LIN {X 0,Y 418.246,Z 523.195,A -85,B 0,C 180,E1 -10027.223,E2 -10027.223} C_VEL
LIN {X 0,Y 418.265,Z 523.195,A -85,B 0,C 180,E1 -10029.679,E2 -10029.679} C_VEL
LIN {X 0,Y 418.284,Z 523.194,A -85,B 0,C 180,E1 -10032.329,E2 -10032.329} C_VEL
LIN {X 0,Y 418.251,Z 523.194,A -85,B 0,C 180,E1 -10035.11,E2 -10035.11} C_VEL
LIN {X 0,Y 418.238,Z 523.199,A -85,B 0,C 180,E1 -10037.766,E2 -10037.766} C_VEL
LIN {X 0,Y 418.257,Z 523.195,A -85,B 0,C 180,E1 -10040.617,E2 -10040.617} C_VEL
LIN {X 0,Y 418.242,Z 523.2,A -85,B 0,C 180,E1 -10043.975,E2 -10043.975} C_VEL
LIN {X 0,Y 418.256,Z 523.193,A -85,B 0,C 180,E1 -10047.155,E2 -10047.155} C_VEL
LIN {X 0,Y 418.27,Z 523.193,A -85,B 0,C 180,E1 -10050.838,E2 -10050.838} C_VEL
LIN {X 0,Y 418.266,Z 523.197,A -85,B 0,C 180,E1 -10054.095,E2 -10054.095} C_VEL
LIN {X 0,Y 418.232,Z 523.196,A -85,B 0,C 180,E1 -10057.263,E2 -10057.263} C_VEL
LIN {X 0,Y 418.309,Z 523.194,A -85,B 0,C 180,E1 -10060.365,E2 -10060.365} C_VEL
LIN {X 0,Y 418.31,Z 523.186,A -85,B 0,C 180,E1 -10063.404,E2 -10063.404} C_VEL
LIN {X 0,Y 418.348,Z 523.183,A -85,B 0,C 180,E1 -10066.993,E2 -10066.993} C_VEL
LIN {X 0,Y 418.352,Z 523.188,A -85,B 0,C 180,E1 -10070.328,E2 -10070.328} C_VEL
LIN {X 0,Y 418.488,Z 523.165,A -85,B 0,C 180,E1 -10073.249,E2 -10073.249} C_VEL
LIN {X 0,Y 418.336,Z 523.184,A -85,B 0,C 180,E1 -10075.181,E2 -10075.181} C_VEL
LIN {X 0,Y 418.536,Z 523.161,A -85,B 0,C 180,E1 -10078.075,E2 -10078.075} C_VEL
LIN {X 0,Y 418.664,Z 523.144,A -85,B 0,C 180,E1 -10080,E2 -10080} C_VEL
LIN {X 0,Y 418.503,Z 523.165,A -85,B 0,C 180,E1 -10082.887,E2 -10082.887} C_VEL
LIN {X 0,Y 418.484,Z 523.17,A -85,B 0,C 180,E1 -10086.751,E2 -10086.751} C_VEL
LIN {X 0,Y 418.333,Z 523.184,A -85,B 0,C 180,E1 -10089.671,E2 -10089.671} C_VEL
LIN {X 0,Y 418.338,Z 523.186,A -85,B 0,C 180,E1 -10093.001,E2 -10093.001} C_VEL
LIN {X 0,Y 418.304,Z 523.193,A -85,B 0,C 180,E1 -10096.735,E2 -10096.735} C_VEL
LIN {X 0,Y 418.262,Z 523.193,A -85,B 0,C 180,E1 -10099.79,E2 -10099.79} C_VEL
LIN {X 0,Y 418.224,Z 523.204,A -85,B 0,C 180,E1 -10102.737,E2 -10102.737} C_VEL
LIN {X 0,Y 418.264,Z 523.193,A -85,B 0,C 180,E1 -10105.904,E2 -10105.904} C_VEL
LIN {X 0,Y 418.267,Z 523.194,A -85,B 0,C 180,E1 -10109.161,E2 -10109.161} C_VEL
LIN {X 0,Y 418.251,Z 523.201,A -85,B 0,C 180,E1 -10112.844,E2 -10112.844} C_VEL
LIN {X 0,Y 418.242,Z 523.197,A -85,B 0,C 180,E1 -10116.239,E2 -10116.239} C_VEL
LIN {X 0,Y 418.243,Z 523.195,A -85,B 0,C 180,E1 -10119.683,E2 -10119.683} C_VEL
LIN {X 0,Y 418.226,Z 523.199,A -85,B 0,C 180,E1 -10122.322,E2 -10122.322} C_VEL
LIN {X 0,Y 418.237,Z 523.2,A -85,B 0,C 180,E1 -10125.11,E2 -10125.11} C_VEL
LIN {X 0,Y 418.237,Z 523.196,A -85,B 0,C 180,E1 -10127.768,E2 -10127.768} C_VEL
LIN {X 0,Y 418.257,Z 523.197,A -85,B 0,C 180,E1 -10130.618,E2 -10130.618} C_VEL
LIN {X 0,Y 418.242,Z 523.198,A -85,B 0,C 180,E1 -10133.977,E2 -10133.977} C_VEL
LIN {X 0,Y 418.289,Z 523.293,A -85,B 0,C 180,E1 -10137.419,E2 -10137.419} C_VEL
LIN {X 0,Y 420.819,Z 535.89,A -85,B 0,C 180,E1 -10140.277,E2 -10140.277} C_VEL
LIN {X 0,Y 421.671,Z 540.942,A -85,B 0,C 180,E1 -10141.369,E2 -10141.369} C_VEL
LIN {X 0,Y 420.647,Z 556.186,A -85,B 0,C 180,E1 -10144.45,E2 -10144.45} C_VEL
LIN {X 0,Y 419.567,Z 573.369,A -85,B 0,C 180,E1 -10147.859,E2 -10147.859} C_VEL
LIN {X 0,Y 418.63,Z 591.451,A -85,B 0,C 180,E1 -10151.4,E2 -10151.4} C_VEL
LIN {X 0,Y 418.074,Z 608.535,A -85,B 0,C 180,E1 -10154.679,E2 -10154.679} C_VEL
LIN {X 0,Y 418.598,Z 615.09,A -85,B 0,C 180,E1 -10154.87,E2 -10154.87} C_VEL
LIN {X 0,Y 421.086,Z 645.701,A -85,B 0,C 180,E1 -10155.582,E2 -10155.582} C_VEL
LIN {X 0,Y 420.445,Z 691.392,A -85,B 0,C 180,E1 -10156.528,E2 -10156.528} C_VEL
LIN {X 0,Y 420.006,Z 702.858,A -85,B 0,C 180,E1 -10156.945,E2 -10156.945} C_VEL
LIN {X 0,Y 419.481,Z 713.993,A -85,B 0,C 180,E1 -10157.543,E2 -10157.543} C_VEL
LIN {X 0,Y 419.018,Z 724.06,A -85,B 0,C 180,E1 -10158.266,E2 -10158.266} C_VEL
LIN {X 0,Y 418.357,Z 734.406,A -85,B 0,C 180,E1 -10159.229,E2 -10159.229} C_VEL
LIN {X 0,Y 417.922,Z 743.55,A -85,B 0,C 180,E1 -10160.319,E2 -10160.319} C_VEL
LIN {X 0,Y 417.662,Z 751.66,A -85,B 0,C 180,E1 -10161.533,E2 -10161.533} C_VEL
LIN {X 0,Y 417.518,Z 759.222,A -85,B 0,C 180,E1 -10162.99,E2 -10162.99} C_VEL
LIN {X 0,Y 417.509,Z 764.103,A -85,B 0,C 180,E1 -10164.203,E2 -10164.203} C_VEL
LIN {X 0,Y 417.604,Z 768.524,A -85,B 0,C 180,E1 -10165.657,E2 -10165.657} C_VEL
LIN {X 0,Y 417.628,Z 771.567,A -85,B 0,C 180,E1 -10167.106,E2 -10167.106} C_VEL
LIN {X 0,Y 417.642,Z 772.856,A -85,B 0,C 180,E1 -10168.071,E2 -10168.071} C_VEL
LIN {X 0,Y 417.68,Z 773.625,A -85,B 0,C 180,E1 -10169.036,E2 -10169.036} C_VEL
LIN {X 0,Y 417.898,Z 773.875,A -85,B 0,C 180,E1 -10170,E2 -10170} C_VEL
LIN {X 0,Y 417.693,Z 773.527,A -85,B 0,C 180,E1 -10170.964,E2 -10170.964} C_VEL
LIN {X 0,Y 417.659,Z 772.684,A -85,B 0,C 180,E1 -10171.928,E2 -10171.928} C_VEL
LIN {X 0,Y 417.645,Z 771.281,A -85,B 0,C 180,E1 -10172.894,E2 -10172.894} C_VEL
LIN {X 0,Y 417.62,Z 768.145,A -85,B 0,C 180,E1 -10174.343,E2 -10174.343} C_VEL
LIN {X 0,Y 417.55,Z 763.608,A -85,B 0,C 180,E1 -10175.796,E2 -10175.796} C_VEL
LIN {X 0,Y 417.469,Z 757.535,A -85,B 0,C 180,E1 -10177.253,E2 -10177.253} C_VEL
LIN {X 0,Y 417.662,Z 751.07,A -85,B 0,C 180,E1 -10178.467,E2 -10178.467} C_VEL
LIN {X 0,Y 417.931,Z 743.033,A -85,B 0,C 180,E1 -10179.681,E2 -10179.681} C_VEL
LIN {X 0,Y 418.336,Z 733.982,A -85,B 0,C 180,E1 -10180.772,E2 -10180.772} C_VEL
LIN {X 0,Y 418.955,Z 723.944,A -85,B 0,C 180,E1 -10181.735,E2 -10181.735} C_VEL
LIN {X 0,Y 419.563,Z 712.596,A -85,B 0,C 180,E1 -10182.577,E2 -10182.577} C_VEL
LIN {X 0,Y 420.235,Z 700.555,A -85,B 0,C 180,E1 -10183.232,E2 -10183.232} C_VEL
LIN {X 0,Y 420.7,Z 688.731,A -85,B 0,C 180,E1 -10183.677,E2 -10183.677} C_VEL
LIN {X 0,Y 420.998,Z 670.166,A -85,B 0,C 180,E1 -10184.081,E2 -10184.081} C_VEL
LIN {X 0,Y 421.223,Z 641.62,A -85,B 0,C 180,E1 -10184.646,E2 -10184.646} C_VEL
LIN {X 0,Y 418.997,Z 611.492,A -85,B 0,C 180,E1 -10185.361,E2 -10185.361} C_VEL
LIN {X 0,Y 417.978,Z 601.746,A -85,B 0,C 180,E1 -10185.637,E2 -10185.637} C_VEL
LIN {X 0,Y 418.254,Z 589.681,A -85,B 0,C 180,E1 -10187.857,E2 -10187.857} C_VEL
LIN {X 0,Y 418.893,Z 571.19,A -85,B 0,C 180,E1 -10191.402,E2 -10191.402} C_VEL
LIN {X 0,Y 419.68,Z 554.188,A -85,B 0,C 180,E1 -10194.749,E2 -10194.749} C_VEL
LIN {X 0,Y 420.676,Z 537.464,A -85,B 0,C 180,E1 -10198.161,E2 -10198.161} C_VEL
LIN {X 0,Y 419.653,Z 530.197,A -85,B 0,C 180,E1 -10199.772,E2 -10199.772} C_VEL
LIN {X 0,Y 418.307,Z 523.383,A -85,B 0,C 180,E1 -10201.387,E2 -10201.387} C_VEL
LIN {X 0,Y 418.256,Z 523.201,A -85,B 0,C 180,E1 -10204.84,E2 -10204.84} C_VEL
LIN {X 0,Y 418.255,Z 523.198,A -85,B 0,C 180,E1 -10208.44,E2 -10208.44} C_VEL
LIN {X 0,Y 418.218,Z 523.205,A -85,B 0,C 180,E1 -10210.947,E2 -10210.947} C_VEL
LIN {X 0,Y 418.212,Z 523.201,A -85,B 0,C 180,E1 -10213.73,E2 -10213.73} C_VEL
LIN {X 0,Y 418.272,Z 523.195,A -85,B 0,C 180,E1 -10216.457,E2 -10216.457} C_VEL
LIN {X 0,Y 418.261,Z 523.2,A -85,B 0,C 180,E1 -10219.123,E2 -10219.123} C_VEL
LIN {X 0,Y 418.232,Z 523.198,A -85,B 0,C 180,E1 -10222.164,E2 -10222.164} C_VEL
LIN {X 0,Y 418.258,Z 523.197,A -85,B 0,C 180,E1 -10225.419,E2 -10225.419} C_VEL
LIN {X 0,Y 418.216,Z 523.201,A -85,B 0,C 180,E1 -10228.605,E2 -10228.605} C_VEL
LIN {X 0,Y 418.287,Z 523.192,A -85,B 0,C 180,E1 -10231.937,E2 -10231.937} C_VEL
LIN {X 0,Y 418.281,Z 523.196,A -85,B 0,C 180,E1 -10235.162,E2 -10235.162} C_VEL
LIN {X 0,Y 418.225,Z 523.201,A -85,B 0,C 180,E1 -10238.303,E2 -10238.303} C_VEL
LIN {X 0,Y 418.275,Z 523.193,A -85,B 0,C 180,E1 -10241.383,E2 -10241.383} C_VEL
LIN {X 0,Y 418.293,Z 523.193,A -85,B 0,C 180,E1 -10244.406,E2 -10244.406} C_VEL
LIN {X 0,Y 418.362,Z 523.185,A -85,B 0,C 180,E1 -10247.386,E2 -10247.386} C_VEL
LIN {X 0,Y 418.352,Z 523.187,A -85,B 0,C 180,E1 -10250.329,E2 -10250.329} C_VEL
LIN {X 0,Y 418.487,Z 523.172,A -85,B 0,C 180,E1 -10253.249,E2 -10253.249} C_VEL
LIN {X 0,Y 418.339,Z 523.189,A -85,B 0,C 180,E1 -10255.182,E2 -10255.182} C_VEL
LIN {X 0,Y 418.536,Z 523.163,A -85,B 0,C 180,E1 -10258.076,E2 -10258.076} C_VEL
LIN {X 0,Y 418.665,Z 523.148,A -85,B 0,C 180,E1 -10260,E2 -10260} C_VEL
LIN {X 0,Y 418.506,Z 523.17,A -85,B 0,C 180,E1 -10262.888,E2 -10262.888} C_VEL
LIN {X 0,Y 418.367,Z 523.437,A -85,B 0,C 180,E1 -10263.552,E2 -10263.552} C_VEL
LIN {X 0,Y 418.557,Z 524.339,A -85,B 0,C 180,E1 -10263.686,E2 -10263.686} C_VEL
LIN {X 0,Y 422.799,Z 535.67,A -85,B 0,C 180,E1 -10264.106,E2 -10264.106} C_VEL
LIN {X 0,Y 422.859,Z 558.987,A -85,B 0,C 180,E1 -10264.56,E2 -10264.56} C_VEL
LIN {X 0,Y 422.802,Z 571.908,A -85,B 0,C 180,E1 -10265.007,E2 -10265.007} C_VEL
LIN {X 0,Y 422.597,Z 583.731,A -85,B 0,C 180,E1 -10265.607,E2 -10265.607} C_VEL
LIN {X 0,Y 422.173,Z 595.975,A -85,B 0,C 180,E1 -10266.452,E2 -10266.452} C_VEL
LIN {X 0,Y 421.729,Z 606.812,A -85,B 0,C 180,E1 -10267.421,E2 -10267.421} C_VEL
LIN {X 0,Y 421.248,Z 615.571,A -85,B 0,C 180,E1 -10268.395,E2 -10268.395} C_VEL
LIN {X 0,Y 420.675,Z 625.172,A -85,B 0,C 180,E1 -10269.716,E2 -10269.716} C_VEL
LIN {X 0,Y 420.062,Z 633.231,A -85,B 0,C 180,E1 -10271.094,E2 -10271.094} C_VEL
LIN {X 0,Y 419.579,Z 640.053,A -85,B 0,C 180,E1 -10272.577,E2 -10272.577} C_VEL
LIN {X 0,Y 419.136,Z 645.457,A -85,B 0,C 180,E1 -10274.072,E2 -10274.072} C_VEL
LIN {X 0,Y 418.765,Z 649.612,A -85,B 0,C 180,E1 -10275.577,E2 -10275.577} C_VEL
LIN {X 0,Y 418.502,Z 652.162,A -85,B 0,C 180,E1 -10276.826,E2 -10276.826} C_VEL
LIN {X 0,Y 418.315,Z 654.541,A -85,B 0,C 180,E1 -10278.616,E2 -10278.616} C_VEL
LIN {X 0,Y 418.2,Z 655.281,A -85,B 0,C 180,E1 -10279.767,E2 -10279.767} C_VEL
LIN {X 0,Y 418.12,Z 655.475,A -85,B 0,C 180,E1 -10280.67,E2 -10280.67} C_VEL
LIN {X 0,Y 418.12,Z 654.832,A -85,B 0,C 180,E1 -10282.415,E2 -10282.415} C_VEL
LIN {X 0,Y 418.179,Z 653.362,A -85,B 0,C 180,E1 -10283.788,E2 -10283.788} C_VEL
LIN {X 0,Y 418.365,Z 650.627,A -85,B 0,C 180,E1 -10285.364,E2 -10285.364} C_VEL
LIN {X 0,Y 418.644,Z 645.998,A -85,B 0,C 180,E1 -10287.162,E2 -10287.162} C_VEL
LIN {X 0,Y 418.944,Z 640.151,A -85,B 0,C 180,E1 -10288.836,E2 -10288.836} C_VEL
LIN {X 0,Y 419.387,Z 632.7,A -85,B 0,C 180,E1 -10290.46,E2 -10290.46} C_VEL
LIN {X 0,Y 419.87,Z 625.218,A -85,B 0,C 180,E1 -10291.765,E2 -10291.765} C_VEL
LIN {X 0,Y 420.353,Z 616.049,A -85,B 0,C 180,E1 -10293.064,E2 -10293.064} C_VEL
LIN {X 0,Y 420.845,Z 605.083,A -85,B 0,C 180,E1 -10294.307,E2 -10294.307} C_VEL
LIN {X 0,Y 421.358,Z 594.46,A -85,B 0,C 180,E1 -10295.262,E2 -10295.262} C_VEL
LIN {X 0,Y 421.75,Z 582.186,A -85,B 0,C 180,E1 -10296.121,E2 -10296.121} C_VEL
LIN {X 0,Y 422,Z 570.008,A -85,B 0,C 180,E1 -10296.763,E2 -10296.763} C_VEL
LIN {X 0,Y 422.095,Z 556.924,A -85,B 0,C 180,E1 -10297.237,E2 -10297.237} C_VEL
LIN {X 0,Y 421.971,Z 535.005,A -85,B 0,C 180,E1 -10297.693,E2 -10297.693} C_VEL
LIN {X 0,Y 418.457,Z 524.063,A -85,B 0,C 180,E1 -10298.046,E2 -10298.046} C_VEL
LIN {X 0,Y 418.305,Z 523.272,A -85,B 0,C 180,E1 -10298.228,E2 -10298.228} C_VEL
LIN {X 0,Y 418.221,Z 523.204,A -85,B 0,C 180,E1 -10300.949,E2 -10300.949} C_VEL
LIN {X 0,Y 418.214,Z 523.204,A -85,B 0,C 180,E1 -10303.732,E2 -10303.732} C_VEL
LIN {X 0,Y 418.266,Z 523.192,A -85,B 0,C 180,E1 -10306.457,E2 -10306.457} C_VEL
LIN {X 0,Y 418.266,Z 523.196,A -85,B 0,C 180,E1 -10309.124,E2 -10309.124} C_VEL
LIN {X 0,Y 418.237,Z 523.196,A -85,B 0,C 180,E1 -10312.166,E2 -10312.166} C_VEL
LIN {X 0,Y 418.265,Z 523.2,A -85,B 0,C 180,E1 -10315.421,E2 -10315.421} C_VEL
LIN {X 0,Y 418.212,Z 523.199,A -85,B 0,C 180,E1 -10318.605,E2 -10318.605} C_VEL
LIN {X 0,Y 418.293,Z 523.191,A -85,B 0,C 180,E1 -10321.938,E2 -10321.938} C_VEL
LIN {X 0,Y 418.292,Z 523.192,A -85,B 0,C 180,E1 -10325.164,E2 -10325.164} C_VEL
LIN {X 0,Y 418.237,Z 523.196,A -85,B 0,C 180,E1 -10328.304,E2 -10328.304} C_VEL
LIN {X 0,Y 418.279,Z 523.195,A -85,B 0,C 180,E1 -10331.383,E2 -10331.383} C_VEL
LIN {X 0,Y 418.306,Z 523.187,A -85,B 0,C 180,E1 -10334.407,E2 -10334.407} C_VEL
LIN {X 0,Y 418.36,Z 523.185,A -85,B 0,C 180,E1 -10337.386,E2 -10337.386} C_VEL
LIN {X 0,Y 418.352,Z 523.181,A -85,B 0,C 180,E1 -10340.708,E2 -10340.708} C_VEL
LIN {X 0,Y 418.464,Z 523.17,A -85,B 0,C 180,E1 -10343.249,E2 -10343.249} C_VEL
LIN {X 0,Y 418.376,Z 523.179,A -85,B 0,C 180,E1 -10344.89,E2 -10344.89} C_VEL
LIN {X 0,Y 417.634,Z 523.279,A -85,B 0,C 180,E1 -10345.694,E2 -10345.694} C_VEL
LIN {X 0,Y 414.774,Z 523.631,A -85,B 0,C 180,E1 -10347.002,E2 -10347.002} C_VEL
LIN {X 0,Y 412.448,Z 523.92,A -85,B 0,C 180,E1 -10348.058,E2 -10348.058} C_VEL
LIN {X 0,Y 411.518,Z 524.034,A -85,B 0,C 180,E1 -10348.874,E2 -10348.874} C_VEL
LIN {X 0,Y 411.476,Z 524.038,A -85,B 0,C 180,E1 -10349.149,E2 -10349.149} C_VEL
LIN {X 0,Y 411.645,Z 524.021,A -85,B 0,C 180,E1 -10350,E2 -10350} C_VEL
LIN {X 0,Y 411.462,Z 524.04,A -85,B 0,C 180,E1 -10352.937,E2 -10352.937} C_VEL
LIN {X 0,Y 411.428,Z 524.044,A -85,B 0,C 180,E1 -10356.867,E2 -10356.867} C_VEL
LIN {X 0,Y 411.297,Z 524.068,A -85,B 0,C 180,E1 -10359.838,E2 -10359.838} C_VEL
LIN {X 0,Y 411.31,Z 524.059,A -85,B 0,C 180,E1 -10363.104,E2 -10363.104} C_VEL
LIN {X 0,Y 411.261,Z 524.065,A -85,B 0,C 180,E1 -10366.888,E2 -10366.888} C_VEL
LIN {X 0,Y 411.234,Z 524.075,A -85,B 0,C 180,E1 -10369.986,E2 -10369.986} C_VEL
LIN {X 0,Y 411.198,Z 524.073,A -85,B 0,C 180,E1 -10373.147,E2 -10373.147} C_VEL
LIN {X 0,Y 411.239,Z 524.07,A -85,B 0,C 180,E1 -10376.38,E2 -10376.38} C_VEL
LIN {X 0,Y 411.202,Z 524.076,A -85,B 0,C 180,E1 -10379.712,E2 -10379.712} C_VEL
LIN {X 0,Y 411.207,Z 524.071,A -85,B 0,C 180,E1 -10383.155,E2 -10383.155} C_VEL
LIN {X 0,Y 411.195,Z 524.075,A -85,B 0,C 180,E1 -10386.552,E2 -10386.552} C_VEL
LIN {X 0,Y 411.227,Z 524.072,A -85,B 0,C 180,E1 -10389.729,E2 -10389.729} C_VEL
LIN {X 0,Y 411.224,Z 524.069,A -85,B 0,C 180,E1 -10393.126,E2 -10393.126} C_VEL
LIN {X 0,Y 411.172,Z 524.08,A -85,B 0,C 180,E1 -10395.879,E2 -10395.879} C_VEL
LIN {X 0,Y 411.162,Z 524.078,A -85,B 0,C 180,E1 -10398.771,E2 -10398.771} C_VEL
LIN {X 0,Y 411.208,Z 524.075,A -85,B 0,C 180,E1 -10401.829,E2 -10401.829} C_VEL
LIN {X 0,Y 411.207,Z 524.071,A -85,B 0,C 180,E1 -10405.12,E2 -10405.12} C_VEL
LIN {X 0,Y 411.168,Z 524.081,A -85,B 0,C 180,E1 -10408.002,E2 -10408.002} C_VEL
LIN {X 0,Y 411.219,Z 524.07,A -85,B 0,C 180,E1 -10411.41,E2 -10411.41} C_VEL
LIN {X 0,Y 411.231,Z 524.071,A -85,B 0,C 180,E1 -10414.706,E2 -10414.706} C_VEL
LIN {X 0,Y 411.199,Z 524.075,A -85,B 0,C 180,E1 -10417.913,E2 -10417.913} C_VEL
LIN {X 0,Y 411.229,Z 524.069,A -85,B 0,C 180,E1 -10421.051,E2 -10421.051} C_VEL
LIN {X 0,Y 411.248,Z 524.071,A -85,B 0,C 180,E1 -10424.131,E2 -10424.131} C_VEL
LIN {X 0,Y 411.307,Z 524.059,A -85,B 0,C 180,E1 -10427.165,E2 -10427.165} C_VEL
LIN {X 0,Y 411.3,Z 524.064,A -85,B 0,C 180,E1 -10430.161,E2 -10430.161} C_VEL
LIN {X 0,Y 411.454,Z 524.041,A -85,B 0,C 180,E1 -10433.133,E2 -10433.133} C_VEL
LIN {X 0,Y 411.307,Z 524.06,A -85,B 0,C 180,E1 -10435.099,E2 -10435.099} C_VEL
LIN {X 0,Y 411.506,Z 524.037,A -85,B 0,C 180,E1 -10438.042,E2 -10438.042} C_VEL
LIN {X 0,Y 411.633,Z 524.02,A -85,B 0,C 180,E1 -10440,E2 -10440} C_VEL
LIN {X 0,Y 411.459,Z 524.043,A -85,B 0,C 180,E1 -10442.937,E2 -10442.937} C_VEL
LIN {X 0,Y 411.448,Z 524.045,A -85,B 0,C 180,E1 -10446.867,E2 -10446.867} C_VEL
LIN {X 0,Y 411.285,Z 524.062,A -85,B 0,C 180,E1 -10449.839,E2 -10449.839} C_VEL
LIN {X 0,Y 411.297,Z 524.062,A -85,B 0,C 180,E1 -10453.104,E2 -10453.104} C_VEL
LIN {X 0,Y 411.255,Z 524.07,A -85,B 0,C 180,E1 -10456.869,E2 -10456.869} C_VEL
LIN {X 0,Y 411.222,Z 524.07,A -85,B 0,C 180,E1 -10459.987,E2 -10459.987} C_VEL
LIN {X 0,Y 411.189,Z 524.076,A -85,B 0,C 180,E1 -10463.148,E2 -10463.148} C_VEL
LIN {X 0,Y 411.231,Z 524.072,A -85,B 0,C 180,E1 -10466.381,E2 -10466.381} C_VEL
LIN {X 0,Y 411.204,Z 524.072,A -85,B 0,C 180,E1 -10469.712,E2 -10469.712} C_VEL
LIN {X 0,Y 411.2,Z 524.075,A -85,B 0,C 180,E1 -10473.156,E2 -10473.156} C_VEL
LIN {X 0,Y 411.189,Z 524.078,A -85,B 0,C 180,E1 -10476.553,E2 -10476.553} C_VEL
LIN {X 0,Y 411.207,Z 524.071,A -85,B 0,C 180,E1 -10479.728,E2 -10479.728} C_VEL
LIN {X 0,Y 411.172,Z 524.08,A -85,B 0,C 180,E1 -10483.133,E2 -10483.133} C_VEL
LIN {X 0,Y 411.168,Z 524.076,A -85,B 0,C 180,E1 -10485.881,E2 -10485.881} C_VEL
LIN {X 0,Y 411.161,Z 524.083,A -85,B 0,C 180,E1 -10488.772,E2 -10488.772} C_VEL
LIN {X 0,Y 411.208,Z 524.071,A -85,B 0,C 180,E1 -10491.831,E2 -10491.831} C_VEL
LIN {X 0,Y 411.208,Z 524.079,A -85,B 0,C 180,E1 -10495.122,E2 -10495.122} C_VEL
LIN {X 0,Y 411.25,Z 524.188,A -85,B 0,C 180,E1 -10497.214,E2 -10497.214} C_VEL
LIN {X 0,Y 413.832,Z 536.994,A -85,B 0,C 180,E1 -10500.172,E2 -10500.172} C_VEL
LIN {X 0,Y 414.674,Z 542.572,A -85,B 0,C 180,E1 -10501.394,E2 -10501.394} C_VEL
LIN {X 0,Y 413.378,Z 560.691,A -85,B 0,C 180,E1 -10505.116,E2 -10505.116} C_VEL
LIN {X 0,Y 412.159,Z 580.028,A -85,B 0,C 180,E1 -10509.018,E2 -10509.018} C_VEL
LIN {X 0,Y 411.367,Z 596.738,A -85,B 0,C 180,E1 -10512.347,E2 -10512.347} C_VEL
LIN {X 0,Y 411.047,Z 607.282,A -85,B 0,C 180,E1 -10514.41,E2 -10514.41} C_VEL
LIN {X 0,Y 411.473,Z 612.884,A -85,B 0,C 180,E1 -10514.585,E2 -10514.585} C_VEL
LIN {X 0,Y 414.19,Z 644.753,A -85,B 0,C 180,E1 -10515.357,E2 -10515.357} C_VEL
LIN {X 0,Y 413.527,Z 690.479,A -85,B 0,C 180,E1 -10516.33,E2 -10516.33} C_VEL
LIN {X 0,Y 413.101,Z 701.187,A -85,B 0,C 180,E1 -10516.722,E2 -10516.722} C_VEL
LIN {X 0,Y 412.539,Z 712.485,A -85,B 0,C 180,E1 -10517.33,E2 -10517.33} C_VEL
LIN {X 0,Y 412.029,Z 722.664,A -85,B 0,C 180,E1 -10518.064,E2 -10518.064} C_VEL
LIN {X 0,Y 411.384,Z 733.084,A -85,B 0,C 180,E1 -10519.044,E2 -10519.044} C_VEL
LIN {X 0,Y 410.895,Z 742.296,A -85,B 0,C 180,E1 -10520.152,E2 -10520.152} C_VEL
LIN {X 0,Y 410.588,Z 750.457,A -85,B 0,C 180,E1 -10521.386,E2 -10521.386} C_VEL
LIN {X 0,Y 410.451,Z 758.066,A -85,B 0,C 180,E1 -10522.869,E2 -10522.869} C_VEL
LIN {X 0,Y 410.465,Z 762.994,A -85,B 0,C 180,E1 -10524.104,E2 -10524.104} C_VEL
LIN {X 0,Y 410.534,Z 767.44,A -85,B 0,C 180,E1 -10525.582,E2 -10525.582} C_VEL
LIN {X 0,Y 410.59,Z 770.518,A -85,B 0,C 180,E1 -10527.057,E2 -10527.057} C_VEL
LIN {X 0,Y 410.606,Z 771.821,A -85,B 0,C 180,E1 -10528.038,E2 -10528.038} C_VEL
LIN {X 0,Y 410.648,Z 772.608,A -85,B 0,C 180,E1 -10529.019,E2 -10529.019} C_VEL
LIN {X 0,Y 410.873,Z 772.863,A -85,B 0,C 180,E1 -10530,E2 -10530} C_VEL
LIN {X 0,Y 410.657,Z 772.53,A -85,B 0,C 180,E1 -10530.981,E2 -10530.981} C_VEL
LIN {X 0,Y 410.617,Z 771.685,A -85,B 0,C 180,E1 -10531.962,E2 -10531.962} C_VEL
LIN {X 0,Y 410.598,Z 770.295,A -85,B 0,C 180,E1 -10532.943,E2 -10532.943} C_VEL
LIN {X 0,Y 410.551,Z 767.157,A -85,B 0,C 180,E1 -10534.418,E2 -10534.418} C_VEL
LIN {X 0,Y 410.499,Z 762.637,A -85,B 0,C 180,E1 -10535.896,E2 -10535.896} C_VEL
LIN {X 0,Y 410.398,Z 756.561,A -85,B 0,C 180,E1 -10537.379,E2 -10537.379} C_VEL
LIN {X 0,Y 410.588,Z 750.109,A -85,B 0,C 180,E1 -10538.613,E2 -10538.613} C_VEL
LIN {X 0,Y 410.9,Z 742.119,A -85,B 0,C 180,E1 -10539.848,E2 -10539.848} C_VEL
LIN {X 0,Y 411.362,Z 733.158,A -85,B 0,C 180,E1 -10540.956,E2 -10540.956} C_VEL
LIN {X 0,Y 411.983,Z 723.228,A -85,B 0,C 180,E1 -10541.937,E2 -10541.937} C_VEL
LIN {X 0,Y 412.63,Z 712.031,A -85,B 0,C 180,E1 -10542.792,E2 -10542.792} C_VEL
LIN {X 0,Y 413.33,Z 700.283,A -85,B 0,C 180,E1 -10543.458,E2 -10543.458} C_VEL
LIN {X 0,Y 413.866,Z 688.335,A -85,B 0,C 180,E1 -10543.93,E2 -10543.93} C_VEL
LIN {X 0,Y 414.156,Z 672.434,A -85,B 0,C 180,E1 -10544.298,E2 -10544.298} C_VEL
LIN {X 0,Y 414.374,Z 641.515,A -85,B 0,C 180,E1 -10544.927,E2 -10544.927} C_VEL
LIN {X 0,Y 412.196,Z 611.847,A -85,B 0,C 180,E1 -10545.654,E2 -10545.654} C_VEL
LIN {X 0,Y 410.931,Z 600.123,A -85,B 0,C 180,E1 -10545.996,E2 -10545.996} C_VEL
LIN {X 0,Y 411.118,Z 592.471,A -85,B 0,C 180,E1 -10547.407,E2 -10547.407} C_VEL
LIN {X 0,Y 411.81,Z 572.728,A -85,B 0,C 180,E1 -10551.263,E2 -10551.263} C_VEL
LIN {X 0,Y 412.602,Z 555.802,A -85,B 0,C 180,E1 -10554.665,E2 -10554.665} C_VEL
LIN {X 0,Y 413.679,Z 539.263,A -85,B 0,C 180,E1 -10558.107,E2 -10558.107} C_VEL
LIN {X 0,Y 413.159,Z 534.02,A -85,B 0,C 180,E1 -10559.277,E2 -10559.277} C_VEL
LIN {X 0,Y 411.25,Z 524.18,A -85,B 0,C 180,E1 -10561.658,E2 -10561.658} C_VEL
LIN {X 0,Y 411.207,Z 524.079,A -85,B 0,C 180,E1 -10564.878,E2 -10564.878} C_VEL
LIN {X 0,Y 411.206,Z 524.075,A -85,B 0,C 180,E1 -10568.169,E2 -10568.169} C_VEL
LIN {X 0,Y 411.159,Z 524.083,A -85,B 0,C 180,E1 -10571.228,E2 -10571.228} C_VEL
LIN {X 0,Y 411.183,Z 524.078,A -85,B 0,C 180,E1 -10574.488,E2 -10574.488} C_VEL
LIN {X 0,Y 411.225,Z 524.069,A -85,B 0,C 180,E1 -10577.296,E2 -10577.296} C_VEL
LIN {X 0,Y 411.225,Z 524.071,A -85,B 0,C 180,E1 -10580.777,E2 -10580.777} C_VEL
LIN {X 0,Y 411.193,Z 524.073,A -85,B 0,C 180,E1 -10584.471,E2 -10584.471} C_VEL
LIN {X 0,Y 411.165,Z 524.076,A -85,B 0,C 180,E1 -10588.003,E2 -10588.003} C_VEL
LIN {X 0,Y 411.216,Z 524.074,A -85,B 0,C 180,E1 -10591.41,E2 -10591.41} C_VEL
LIN {X 0,Y 411.228,Z 524.072,A -85,B 0,C 180,E1 -10594.707,E2 -10594.707} C_VEL
LIN {X 0,Y 411.197,Z 524.075,A -85,B 0,C 180,E1 -10597.913,E2 -10597.913} C_VEL
LIN {X 0,Y 411.216,Z 524.076,A -85,B 0,C 180,E1 -10601.051,E2 -10601.051} C_VEL
LIN {X 0,Y 411.246,Z 524.07,A -85,B 0,C 180,E1 -10604.132,E2 -10604.132} C_VEL
LIN {X 0,Y 411.306,Z 524.063,A -85,B 0,C 180,E1 -10607.166,E2 -10607.166} C_VEL
LIN {X 0,Y 411.3,Z 524.064,A -85,B 0,C 180,E1 -10610.162,E2 -10610.162} C_VEL
LIN {X 0,Y 411.453,Z 524.048,A -85,B 0,C 180,E1 -10613.133,E2 -10613.133} C_VEL
LIN {X 0,Y 411.311,Z 524.065,A -85,B 0,C 180,E1 -10615.099,E2 -10615.099} C_VEL
LIN {X 0,Y 411.505,Z 524.039,A -85,B 0,C 180,E1 -10618.043,E2 -10618.043} C_VEL
LIN {X 0,Y 411.634,Z 524.024,A -85,B 0,C 180,E1 -10620,E2 -10620} C_VEL
LIN {X 0,Y 411.42,Z 524.223,A -85,B 0,C 180,E1 -10623.183,E2 -10623.183} C_VEL
LIN {X 0,Y 411.562,Z 525.055,A -85,B 0,C 180,E1 -10623.335,E2 -10623.335} C_VEL
LIN {X 0,Y 415.966,Z 536.472,A -85,B 0,C 180,E1 -10623.793,E2 -10623.793} C_VEL
LIN {X 0,Y 416.165,Z 561.028,A -85,B 0,C 180,E1 -10624.298,E2 -10624.298} C_VEL
LIN {X 0,Y 416.077,Z 573.898,A -85,B 0,C 180,E1 -10624.76,E2 -10624.76} C_VEL
LIN {X 0,Y 415.895,Z 584.85,A -85,B 0,C 180,E1 -10625.333,E2 -10625.333} C_VEL
LIN {X 0,Y 415.457,Z 597.105,A -85,B 0,C 180,E1 -10626.191,E2 -10626.191} C_VEL
LIN {X 0,Y 414.968,Z 607.968,A -85,B 0,C 180,E1 -10627.176,E2 -10627.176} C_VEL
LIN {X 0,Y 414.404,Z 617.684,A -85,B 0,C 180,E1 -10628.289,E2 -10628.289} C_VEL
LIN {X 0,Y 413.819,Z 626.75,A -85,B 0,C 180,E1 -10629.577,E2 -10629.577} C_VEL
LIN {X 0,Y 413.135,Z 634.964,A -85,B 0,C 180,E1 -10631.034,E2 -10631.034} C_VEL
LIN {X 0,Y 412.719,Z 640.648,A -85,B 0,C 180,E1 -10632.29,E2 -10632.29} C_VEL
LIN {X 0,Y 412.218,Z 646.149,A -85,B 0,C 180,E1 -10633.81,E2 -10633.81} C_VEL
LIN {X 0,Y 411.814,Z 650.39,A -85,B 0,C 180,E1 -10635.339,E2 -10635.339} C_VEL
LIN {X 0,Y 411.502,Z 653.649,A -85,B 0,C 180,E1 -10636.982,E2 -10636.982} C_VEL
LIN {X 0,Y 411.367,Z 654.936,A -85,B 0,C 180,E1 -10637.91,E2 -10637.91} C_VEL
LIN {X 0,Y 411.255,Z 655.894,A -85,B 0,C 180,E1 -10638.947,E2 -10638.947} C_VEL
LIN {X 0,Y 411.182,Z 656.423,A -85,B 0,C 180,E1 -10639.99,E2 -10639.99} C_VEL
LIN {X 0,Y 411.095,Z 656.474,A -85,B 0,C 180,E1 -10641.04,E2 -10641.04} C_VEL
LIN {X 0,Y 411.109,Z 655.662,A -85,B 0,C 180,E1 -10642.614,E2 -10642.614} C_VEL
LIN {X 0,Y 411.182,Z 653.743,A -85,B 0,C 180,E1 -10644.219,E2 -10644.219} C_VEL
LIN {X 0,Y 411.403,Z 650.665,A -85,B 0,C 180,E1 -10645.825,E2 -10645.825} C_VEL
LIN {X 0,Y 411.672,Z 646.308,A -85,B 0,C 180,E1 -10647.448,E2 -10647.448} C_VEL
LIN {X 0,Y 411.989,Z 640.568,A -85,B 0,C 180,E1 -10649.054,E2 -10649.054} C_VEL
LIN {X 0,Y 412.383,Z 634.18,A -85,B 0,C 180,E1 -10650.465,E2 -10650.465} C_VEL
LIN {X 0,Y 412.89,Z 626.443,A -85,B 0,C 180,E1 -10651.848,E2 -10651.848} C_VEL
LIN {X 0,Y 413.387,Z 617.24,A -85,B 0,C 180,E1 -10653.181,E2 -10653.181} C_VEL
LIN {X 0,Y 413.914,Z 606.962,A -85,B 0,C 180,E1 -10654.373,E2 -10654.373} C_VEL
LIN {X 0,Y 414.433,Z 595.618,A -85,B 0,C 180,E1 -10655.423,E2 -10655.423} C_VEL
LIN {X 0,Y 414.812,Z 584.183,A -85,B 0,C 180,E1 -10656.246,E2 -10656.246} C_VEL
LIN {X 0,Y 415.129,Z 571.393,A -85,B 0,C 180,E1 -10656.941,E2 -10656.941} C_VEL
LIN {X 0,Y 415.221,Z 558.345,A -85,B 0,C 180,E1 -10657.429,E2 -10657.429} C_VEL
LIN {X 0,Y 415.242,Z 538.876,A -85,B 0,C 180,E1 -10657.849,E2 -10657.849} C_VEL
LIN {X 0,Y 414.968,Z 535.994,A -85,B 0,C 180,E1 -10657.914,E2 -10657.914} C_VEL
LIN {X 0,Y 411.405,Z 524.965,A -85,B 0,C 180,E1 -10658.278,E2 -10658.278} C_VEL
LIN {X 0,Y 411.253,Z 524.149,A -85,B 0,C 180,E1 -10658.467,E2 -10658.467} C_VEL
LIN {X 0,Y 411.176,Z 524.08,A -85,B 0,C 180,E1 -10661.806,E2 -10661.806} C_VEL
LIN {X 0,Y 411.223,Z 524.075,A -85,B 0,C 180,E1 -10665.517,E2 -10665.517} C_VEL
LIN {X 0,Y 411.208,Z 524.072,A -85,B 0,C 180,E1 -10668.765,E2 -10668.765} C_VEL
LIN {X 0,Y 411.203,Z 524.073,A -85,B 0,C 180,E1 -10672.028,E2 -10672.028} C_VEL
LIN {X 0,Y 411.206,Z 524.076,A -85,B 0,C 180,E1 -10675.667,E2 -10675.667} C_VEL
LIN {X 0,Y 411.19,Z 524.077,A -85,B 0,C 180,E1 -10679.153,E2 -10679.153} C_VEL
LIN {X 0,Y 411.261,Z 524.065,A -85,B 0,C 180,E1 -10682.523,E2 -10682.523} C_VEL
LIN {X 0,Y 411.23,Z 524.073,A -85,B 0,C 180,E1 -10685.785,E2 -10685.785} C_VEL
LIN {X 0,Y 411.199,Z 524.074,A -85,B 0,C 180,E1 -10688.967,E2 -10688.967} C_VEL
LIN {X 0,Y 411.249,Z 524.068,A -85,B 0,C 180,E1 -10692.085,E2 -10692.085} C_VEL
LIN {X 0,Y 411.264,Z 524.066,A -85,B 0,C 180,E1 -10695.148,E2 -10695.148} C_VEL
LIN {X 0,Y 411.287,Z 524.063,A -85,B 0,C 180,E1 -10698.168,E2 -10698.168} C_VEL
LIN {X 0,Y 411.356,Z 524.055,A -85,B 0,C 180,E1 -10701.155,E2 -10701.155} C_VEL
LIN {X 0,Y 411.447,Z 524.044,A -85,B 0,C 180,E1 -10704.118,E2 -10704.118} C_VEL
LIN {X 0,Y 411.516,Z 524.036,A -85,B 0,C 180,E1 -10708.043,E2 -10708.043} C_VEL
LIN {X 0,Y 411.476,Z 524.038,A -85,B 0,C 180,E1 -10709.149,E2 -10709.149} C_VEL
LIN {X 0,Y 410.908,Z 524.113,A -85,B 0,C 180,E1 -10709.967,E2 -10709.967} C_VEL
LIN {X 0,Y 408.098,Z 524.461,A -85,B 0,C 180,E1 -10711.296,E2 -10711.296} C_VEL
LIN {X 0,Y 405.6,Z 524.771,A -85,B 0,C 180,E1 -10712.369,E2 -10712.369} C_VEL
LIN {X 0,Y 404.437,Z 524.916,A -85,B 0,C 180,E1 -10713.199,E2 -10713.199} C_VEL
LIN {X 0,Y 404.297,Z 524.933,A -85,B 0,C 180,E1 -10713.481,E2 -10713.481} C_VEL
LIN {X 0,Y 404.397,Z 524.925,A -85,B 0,C 180,E1 -10715.985,E2 -10715.985} C_VEL
LIN {X 0,Y 404.271,Z 524.936,A -85,B 0,C 180,E1 -10719.001,E2 -10719.001} C_VEL
LIN {X 0,Y 404.261,Z 524.942,A -85,B 0,C 180,E1 -10722.041,E2 -10722.041} C_VEL
LIN {X 0,Y 404.21,Z 524.943,A -85,B 0,C 180,E1 -10725.118,E2 -10725.118} C_VEL
LIN {X 0,Y 404.214,Z 524.946,A -85,B 0,C 180,E1 -10728.238,E2 -10728.238} C_VEL
LIN {X 0,Y 404.142,Z 524.953,A -85,B 0,C 180,E1 -10731.419,E2 -10731.419} C_VEL
LIN {X 0,Y 404.176,Z 524.948,A -85,B 0,C 180,E1 -10734.665,E2 -10734.665} C_VEL
LIN {X 0,Y 404.197,Z 524.952,A -85,B 0,C 180,E1 -10737.999,E2 -10737.999} C_VEL
LIN {X 0,Y 404.14,Z 524.954,A -85,B 0,C 180,E1 -10741.557,E2 -10741.557} C_VEL
LIN {X 0,Y 404.185,Z 524.946,A -85,B 0,C 180,E1 -10745.015,E2 -10745.015} C_VEL
LIN {X 0,Y 404.163,Z 524.95,A -85,B 0,C 180,E1 -10748.755,E2 -10748.755} C_VEL
LIN {X 0,Y 404.191,Z 524.948,A -85,B 0,C 180,E1 -10751.61,E2 -10751.61} C_VEL
LIN {X 0,Y 404.19,Z 524.948,A -85,B 0,C 180,E1 -10754.528,E2 -10754.528} C_VEL
LIN {X 0,Y 404.135,Z 524.953,A -85,B 0,C 180,E1 -10757.295,E2 -10757.295} C_VEL
LIN {X 0,Y 404.166,Z 524.953,A -85,B 0,C 180,E1 -10759.954,E2 -10759.954} C_VEL
LIN {X 0,Y 404.136,Z 524.952,A -85,B 0,C 180,E1 -10763.123,E2 -10763.123} C_VEL
LIN {X 0,Y 404.141,Z 524.959,A -85,B 0,C 180,E1 -10766.187,E2 -10766.187} C_VEL
LIN {X 0,Y 404.16,Z 524.951,A -85,B 0,C 180,E1 -10769.716,E2 -10769.716} C_VEL
LIN {X 0,Y 404.19,Z 524.946,A -85,B 0,C 180,E1 -10773.122,E2 -10773.122} C_VEL
LIN {X 0,Y 404.171,Z 524.948,A -85,B 0,C 180,E1 -10775.334,E2 -10775.334} C_VEL
LIN {X 0,Y 404.157,Z 524.954,A -85,B 0,C 180,E1 -10778.581,E2 -10778.581} C_VEL
LIN {X 0,Y 404.207,Z 524.945,A -85,B 0,C 180,E1 -10781.761,E2 -10781.761} C_VEL
LIN {X 0,Y 404.2,Z 524.946,A -85,B 0,C 180,E1 -10784.881,E2 -10784.881} C_VEL
LIN {X 0,Y 404.262,Z 524.939,A -85,B 0,C 180,E1 -10787.958,E2 -10787.958} C_VEL
LIN {X 0,Y 404.426,Z 524.92,A -85,B 0,C 180,E1 -10792.099,E2 -10792.099} C_VEL
LIN {X 0,Y 404.419,Z 524.919,A -85,B 0,C 180,E1 -10794.015,E2 -10794.015} C_VEL
LIN {X 0,Y 404.475,Z 524.912,A -85,B 0,C 180,E1 -10798.008,E2 -10798.008} C_VEL
LIN {X 0,Y 404.603,Z 524.896,A -85,B 0,C 180,E1 -10800,E2 -10800} C_VEL
LIN {X 0,Y 404.416,Z 524.919,A -85,B 0,C 180,E1 -10802.988,E2 -10802.988} C_VEL
LIN {X 0,Y 404.394,Z 524.922,A -85,B 0,C 180,E1 -10806.987,E2 -10806.987} C_VEL
LIN {X 0,Y 404.25,Z 524.939,A -85,B 0,C 180,E1 -10810.012,E2 -10810.012} C_VEL
LIN {X 0,Y 404.258,Z 524.938,A -85,B 0,C 180,E1 -10813.211,E2 -10813.211} C_VEL
LIN {X 0,Y 404.208,Z 524.946,A -85,B 0,C 180,E1 -10817.007,E2 -10817.007} C_VEL
LIN {X 0,Y 404.156,Z 524.953,A -85,B 0,C 180,E1 -10820.352,E2 -10820.352} C_VEL
LIN {X 0,Y 404.156,Z 524.95,A -85,B 0,C 180,E1 -10823.575,E2 -10823.575} C_VEL
LIN {X 0,Y 404.176,Z 524.947,A -85,B 0,C 180,E1 -10825.767,E2 -10825.767} C_VEL
LIN {X 0,Y 404.191,Z 524.946,A -85,B 0,C 180,E1 -10828,E2 -10828} C_VEL
LIN {X 0,Y 404.136,Z 524.952,A -85,B 0,C 180,E1 -10831.559,E2 -10831.559} C_VEL
LIN {X 0,Y 404.179,Z 524.951,A -85,B 0,C 180,E1 -10835.016,E2 -10835.016} C_VEL
LIN {X 0,Y 404.15,Z 524.957,A -85,B 0,C 180,E1 -10838.757,E2 -10838.757} C_VEL
LIN {X 0,Y 404.118,Z 524.955,A -85,B 0,C 180,E1 -10841.6,E2 -10841.6} C_VEL
LIN {X 0,Y 404.145,Z 524.955,A -85,B 0,C 180,E1 -10844.523,E2 -10844.523} C_VEL
LIN {X 0,Y 404.134,Z 524.955,A -85,B 0,C 180,E1 -10847.296,E2 -10847.296} C_VEL
LIN {X 0,Y 404.164,Z 524.949,A -85,B 0,C 180,E1 -10849.956,E2 -10849.956} C_VEL
LIN {X 0,Y 404.136,Z 524.958,A -85,B 0,C 180,E1 -10853.125,E2 -10853.125} C_VEL
LIN {X 0,Y 404.15,Z 524.957,A -85,B 0,C 180,E1 -10856.189,E2 -10856.189} C_VEL
LIN {X 0,Y 404.222,Z 525.206,A -85,B 0,C 180,E1 -10857.052,E2 -10857.052} C_VEL
LIN {X 0,Y 406.949,Z 538.808,A -85,B 0,C 180,E1 -10860.231,E2 -10860.231} C_VEL
LIN {X 0,Y 407.649,Z 542.843,A -85,B 0,C 180,E1 -10861.137,E2 -10861.137} C_VEL
LIN {X 0,Y 406.83,Z 554.991,A -85,B 0,C 180,E1 -10863.697,E2 -10863.697} C_VEL
LIN {X 0,Y 405.75,Z 569.651,A -85,B 0,C 180,E1 -10866.738,E2 -10866.738} C_VEL
LIN {X 0,Y 404.726,Z 587.886,A -85,B 0,C 180,E1 -10870.472,E2 -10870.472} C_VEL
LIN {X 0,Y 403.96,Z 606.305,A -85,B 0,C 180,E1 -10874.162,E2 -10874.162} C_VEL
LIN {X 0,Y 405.925,Z 628.91,A -85,B 0,C 180,E1 -10874.755,E2 -10874.755} C_VEL
LIN {X 0,Y 407.225,Z 646.126,A -85,B 0,C 180,E1 -10875.172,E2 -10875.172} C_VEL
LIN {X 0,Y 406.563,Z 689.529,A -85,B 0,C 180,E1 -10876.123,E2 -10876.123} C_VEL
LIN {X 0,Y 406.113,Z 700.859,A -85,B 0,C 180,E1 -10876.553,E2 -10876.553} C_VEL
LIN {X 0,Y 405.564,Z 710.966,A -85,B 0,C 180,E1 -10877.108,E2 -10877.108} C_VEL
LIN {X 0,Y 404.979,Z 721.238,A -85,B 0,C 180,E1 -10877.853,E2 -10877.853} C_VEL
LIN {X 0,Y 404.384,Z 731.755,A -85,B 0,C 180,E1 -10878.852,E2 -10878.852} C_VEL
LIN {X 0,Y 404.005,Z 739.174,A -85,B 0,C 180,E1 -10879.729,E2 -10879.729} C_VEL
LIN {X 0,Y 403.561,Z 747.734,A -85,B 0,C 180,E1 -10880.983,E2 -10880.983} C_VEL
LIN {X 0,Y 403.406,Z 754.584,A -85,B 0,C 180,E1 -10882.24,E2 -10882.24} C_VEL
LIN {X 0,Y 403.401,Z 760.268,A -85,B 0,C 180,E1 -10883.562,E2 -10883.562} C_VEL
LIN {X 0,Y 403.413,Z 765.02,A -85,B 0,C 180,E1 -10885.003,E2 -10885.003} C_VEL
LIN {X 0,Y 403.592,Z 767.554,A -85,B 0,C 180,E1 -10886.006,E2 -10886.006} C_VEL
LIN {X 0,Y 403.55,Z 769.466,A -85,B 0,C 180,E1 -10887.005,E2 -10887.005} C_VEL
LIN {X 0,Y 403.569,Z 770.784,A -85,B 0,C 180,E1 -10888.004,E2 -10888.004} C_VEL
LIN {X 0,Y 403.615,Z 771.591,A -85,B 0,C 180,E1 -10889.002,E2 -10889.002} C_VEL
LIN {X 0,Y 403.847,Z 771.851,A -85,B 0,C 180,E1 -10890,E2 -10890} C_VEL
LIN {X 0,Y 403.621,Z 771.532,A -85,B 0,C 180,E1 -10890.998,E2 -10890.998} C_VEL
LIN {X 0,Y 403.574,Z 770.687,A -85,B 0,C 180,E1 -10891.996,E2 -10891.996} C_VEL
LIN {X 0,Y 403.549,Z 769.305,A -85,B 0,C 180,E1 -10892.995,E2 -10892.995} C_VEL
LIN {X 0,Y 403.483,Z 766.169,A -85,B 0,C 180,E1 -10894.495,E2 -10894.495} C_VEL
LIN {X 0,Y 403.4,Z 761.669,A -85,B 0,C 180,E1 -10896,E2 -10896} C_VEL
LIN {X 0,Y 403.339,Z 755.626,A -85,B 0,C 180,E1 -10897.509,E2 -10897.509} C_VEL
LIN {X 0,Y 403.527,Z 749.229,A -85,B 0,C 180,E1 -10898.765,E2 -10898.765} C_VEL
LIN {X 0,Y 403.88,Z 741.267,A -85,B 0,C 180,E1 -10900.021,E2 -10900.021} C_VEL
LIN {X 0,Y 404.265,Z 733.471,A -85,B 0,C 180,E1 -10901.024,E2 -10901.024} C_VEL
LIN {X 0,Y 404.917,Z 723.86,A -85,B 0,C 180,E1 -10902.021,E2 -10902.021} C_VEL
LIN {X 0,Y 405.602,Z 713.272,A -85,B 0,C 180,E1 -10902.89,E2 -10902.89} C_VEL
LIN {X 0,Y 406.378,Z 701.209,A -85,B 0,C 180,E1 -10903.629,E2 -10903.629} C_VEL
LIN {X 0,Y 406.934,Z 689.008,A -85,B 0,C 180,E1 -10904.152,E2 -10904.152} C_VEL
LIN {X 0,Y 407.293,Z 676.682,A -85,B 0,C 180,E1 -10904.484,E2 -10904.484} C_VEL
LIN {X 0,Y 407.68,Z 642.972,A -85,B 0,C 180,E1 -10905.187,E2 -10905.187} C_VEL
LIN {X 0,Y 405.287,Z 610.498,A -85,B 0,C 180,E1 -10906.011,E2 -10906.011} C_VEL
LIN {X 0,Y 403.927,Z 598.351,A -85,B 0,C 180,E1 -10906.38,E2 -10906.38} C_VEL
LIN {X 0,Y 404.306,Z 583.4,A -85,B 0,C 180,E1 -10909.285,E2 -10909.285} C_VEL
LIN {X 0,Y 404.97,Z 567.747,A -85,B 0,C 180,E1 -10912.444,E2 -10912.444} C_VEL
LIN {X 0,Y 405.915,Z 551.581,A -85,B 0,C 180,E1 -10915.8,E2 -10915.8} C_VEL
LIN {X 0,Y 406.693,Z 538.986,A -85,B 0,C 180,E1 -10918.508,E2 -10918.508} C_VEL
LIN {X 0,Y 405.073,Z 529.362,A -85,B 0,C 180,E1 -10920.784,E2 -10920.784} C_VEL
LIN {X 0,Y 404.183,Z 525.032,A -85,B 0,C 180,E1 -10921.917,E2 -10921.917} C_VEL
LIN {X 0,Y 404.178,Z 524.954,A -85,B 0,C 180,E1 -10925.189,E2 -10925.189} C_VEL
LIN {X 0,Y 404.153,Z 524.955,A -85,B 0,C 180,E1 -10928.756,E2 -10928.756} C_VEL
LIN {X 0,Y 404.119,Z 524.956,A -85,B 0,C 180,E1 -10931.599,E2 -10931.599} C_VEL
LIN {X 0,Y 404.152,Z 524.953,A -85,B 0,C 180,E1 -10934.523,E2 -10934.523} C_VEL
LIN {X 0,Y 404.203,Z 524.944,A -85,B 0,C 180,E1 -10937.305,E2 -10937.305} C_VEL
LIN {X 0,Y 404.162,Z 524.951,A -85,B 0,C 180,E1 -10939.955,E2 -10939.955} C_VEL
LIN {X 0,Y 404.134,Z 524.956,A -85,B 0,C 180,E1 -10943.124,E2 -10943.124} C_VEL
LIN {X 0,Y 404.138,Z 524.955,A -85,B 0,C 180,E1 -10946.187,E2 -10946.187} C_VEL
LIN {X 0,Y 404.148,Z 524.952,A -85,B 0,C 180,E1 -10949.715,E2 -10949.715} C_VEL
LIN {X 0,Y 404.187,Z 524.947,A -85,B 0,C 180,E1 -10953.123,E2 -10953.123} C_VEL
LIN {X 0,Y 404.169,Z 524.952,A -85,B 0,C 180,E1 -10955.334,E2 -10955.334} C_VEL
LIN {X 0,Y 404.151,Z 524.956,A -85,B 0,C 180,E1 -10958.582,E2 -10958.582} C_VEL
LIN {X 0,Y 404.201,Z 524.945,A -85,B 0,C 180,E1 -10961.762,E2 -10961.762} C_VEL
LIN {X 0,Y 404.199,Z 524.948,A -85,B 0,C 180,E1 -10964.882,E2 -10964.882} C_VEL
LIN {X 0,Y 404.263,Z 524.94,A -85,B 0,C 180,E1 -10967.959,E2 -10967.959} C_VEL
LIN {X 0,Y 404.424,Z 524.922,A -85,B 0,C 180,E1 -10972.1,E2 -10972.1} C_VEL
LIN {X 0,Y 404.43,Z 524.92,A -85,B 0,C 180,E1 -10974.016,E2 -10974.016} C_VEL
LIN {X 0,Y 404.474,Z 524.915,A -85,B 0,C 180,E1 -10978.009,E2 -10978.009} C_VEL
LIN {X 0,Y 404.604,Z 524.9,A -85,B 0,C 180,E1 -10980,E2 -10980} C_VEL
LIN {X 0,Y 404.438,Z 525.043,A -85,B 0,C 180,E1 -10982.802,E2 -10982.802} C_VEL
LIN {X 0,Y 404.612,Z 526.038,A -85,B 0,C 180,E1 -10982.987,E2 -10982.987} C_VEL
LIN {X 0,Y 409.4,Z 538.47,A -85,B 0,C 180,E1 -10983.506,E2 -10983.506} C_VEL
LIN {X 0,Y 409.487,Z 561.124,A -85,B 0,C 180,E1 -10983.968,E2 -10983.968} C_VEL
LIN {X 0,Y 409.391,Z 574.417,A -85,B 0,C 180,E1 -10984.442,E2 -10984.442} C_VEL
LIN {X 0,Y 409.202,Z 585.953,A -85,B 0,C 180,E1 -10985.049,E2 -10985.049} C_VEL
LIN {X 0,Y 408.723,Z 598.258,A -85,B 0,C 180,E1 -10985.922,E2 -10985.922} C_VEL
LIN {X 0,Y 408.216,Z 609.124,A -85,B 0,C 180,E1 -10986.922,E2 -10986.922} C_VEL
LIN {X 0,Y 407.683,Z 617.887,A -85,B 0,C 180,E1 -10987.927,E2 -10987.927} C_VEL
LIN {X 0,Y 407.102,Z 626.487,A -85,B 0,C 180,E1 -10989.138,E2 -10989.138} C_VEL
LIN {X 0,Y 406.456,Z 634.163,A -85,B 0,C 180,E1 -10990.461,E2 -10990.461} C_VEL
LIN {X 0,Y 405.87,Z 641.29,A -85,B 0,C 180,E1 -10991.993,E2 -10991.993} C_VEL
LIN {X 0,Y 405.259,Z 647.694,A -85,B 0,C 180,E1 -10993.801,E2 -10993.801} C_VEL
LIN {X 0,Y 404.784,Z 652.379,A -85,B 0,C 180,E1 -10995.612,E2 -10995.612} C_VEL
LIN {X 0,Y 404.465,Z 655.155,A -85,B 0,C 180,E1 -10997.182,E2 -10997.182} C_VEL
LIN {X 0,Y 404.328,Z 656.4,A -85,B 0,C 180,E1 -10998.233,E2 -10998.233} C_VEL
LIN {X 0,Y 404.158,Z 657.507,A -85,B 0,C 180,E1 -11000.116,E2 -11000.116} C_VEL
LIN {X 0,Y 404.082,Z 657.388,A -85,B 0,C 180,E1 -11001.423,E2 -11001.423} C_VEL
LIN {X 0,Y 404.079,Z 656.491,A -85,B 0,C 180,E1 -11002.811,E2 -11002.811} C_VEL
LIN {X 0,Y 404.215,Z 654.067,A -85,B 0,C 180,E1 -11004.664,E2 -11004.664} C_VEL
LIN {X 0,Y 404.466,Z 650.628,A -85,B 0,C 180,E1 -11006.302,E2 -11006.302} C_VEL
LIN {X 0,Y 404.738,Z 645.846,A -85,B 0,C 180,E1 -11007.959,E2 -11007.959} C_VEL
LIN {X 0,Y 405.059,Z 640.223,A -85,B 0,C 180,E1 -11009.465,E2 -11009.465} C_VEL
LIN {X 0,Y 405.545,Z 632.801,A -85,B 0,C 180,E1 -11011.035,E2 -11011.035} C_VEL
LIN {X 0,Y 406.067,Z 624.424,A -85,B 0,C 180,E1 -11012.448,E2 -11012.448} C_VEL
LIN {X 0,Y 406.658,Z 615.159,A -85,B 0,C 180,E1 -11013.717,E2 -11013.717} C_VEL
LIN {X 0,Y 407.117,Z 604.61,A -85,B 0,C 180,E1 -11014.879,E2 -11014.879} C_VEL
LIN {X 0,Y 407.68,Z 593.075,A -85,B 0,C 180,E1 -11015.883,E2 -11015.883} C_VEL
LIN {X 0,Y 408.017,Z 581.102,A -85,B 0,C 180,E1 -11016.691,E2 -11016.691} C_VEL
LIN {X 0,Y 408.266,Z 567.975,A -85,B 0,C 180,E1 -11017.337,E2 -11017.337} C_VEL
LIN {X 0,Y 408.32,Z 555.828,A -85,B 0,C 180,E1 -11017.742,E2 -11017.742} C_VEL
LIN {X 0,Y 408.321,Z 538.067,A -85,B 0,C 180,E1 -11018.104,E2 -11018.104} C_VEL
LIN {X 0,Y 404.393,Z 525.909,A -85,B 0,C 180,E1 -11018.502,E2 -11018.502} C_VEL
LIN {X 0,Y 404.207,Z 525.013,A -85,B 0,C 180,E1 -11018.712,E2 -11018.712} C_VEL
LIN {X 0,Y 404.122,Z 524.961,A -85,B 0,C 180,E1 -11021.601,E2 -11021.601} C_VEL
LIN {X 0,Y 404.154,Z 524.95,A -85,B 0,C 180,E1 -11024.525,E2 -11024.525} C_VEL
LIN {X 0,Y 404.205,Z 524.95,A -85,B 0,C 180,E1 -11027.306,E2 -11027.306} C_VEL
LIN {X 0,Y 404.168,Z 524.95,A -85,B 0,C 180,E1 -11029.956,E2 -11029.956} C_VEL
LIN {X 0,Y 404.14,Z 524.955,A -85,B 0,C 180,E1 -11033.125,E2 -11033.125} C_VEL
LIN {X 0,Y 404.145,Z 524.952,A -85,B 0,C 180,E1 -11036.189,E2 -11036.189} C_VEL
LIN {X 0,Y 404.147,Z 524.956,A -85,B 0,C 180,E1 -11039.716,E2 -11039.716} C_VEL
LIN {X 0,Y 404.197,Z 524.947,A -85,B 0,C 180,E1 -11043.124,E2 -11043.124} C_VEL
LIN {X 0,Y 404.18,Z 524.952,A -85,B 0,C 180,E1 -11045.335,E2 -11045.335} C_VEL
LIN {X 0,Y 404.141,Z 524.951,A -85,B 0,C 180,E1 -11048.581,E2 -11048.581} C_VEL
LIN {X 0,Y 404.208,Z 524.949,A -85,B 0,C 180,E1 -11051.762,E2 -11051.762} C_VEL
LIN {X 0,Y 404.21,Z 524.943,A -85,B 0,C 180,E1 -11054.883,E2 -11054.883} C_VEL
LIN {X 0,Y 404.26,Z 524.94,A -85,B 0,C 180,E1 -11057.959,E2 -11057.959} C_VEL
LIN {X 0,Y 404.293,Z 524.933,A -85,B 0,C 180,E1 -11060.999,E2 -11060.999} C_VEL
LIN {X 0,Y 404.397,Z 524.923,A -85,B 0,C 180,E1 -11064.015,E2 -11064.015} C_VEL
LIN {X 0,Y 404.485,Z 524.913,A -85,B 0,C 180,E1 -11068.009,E2 -11068.009} C_VEL
LIN {X 0,Y 404.615,Z 524.897,A -85,B 0,C 180,E1 -11070,E2 -11070} C_VEL
LIN {X 0,Y 404.42,Z 524.917,A -85,B 0,C 180,E1 -11072.988,E2 -11072.988} C_VEL
LIN {X 0,Y 404.297,Z 524.933,A -85,B 0,C 180,E1 -11073.481,E2 -11073.481} C_VEL
LIN {X 0,Y 403.539,Z 525.032,A -85,B 0,C 180,E1 -11074.312,E2 -11074.312} C_VEL
LIN {X 0,Y 400.76,Z 525.388,A -85,B 0,C 180,E1 -11075.666,E2 -11075.666} C_VEL
LIN {X 0,Y 398.448,Z 525.677,A -85,B 0,C 180,E1 -11076.76,E2 -11076.76} C_VEL
LIN {X 0,Y 397.42,Z 525.799,A -85,B 0,C 180,E1 -11077.603,E2 -11077.603} C_VEL
LIN {X 0,Y 397.311,Z 525.809,A -85,B 0,C 180,E1 -11077.889,E2 -11077.889} C_VEL
LIN {X 0,Y 397.203,Z 525.817,A -85,B 0,C 180,E1 -11081.223,E2 -11081.223} C_VEL
LIN {X 0,Y 397.181,Z 525.821,A -85,B 0,C 180,E1 -11084.343,E2 -11084.343} C_VEL
LIN {X 0,Y 397.178,Z 525.822,A -85,B 0,C 180,E1 -11087.506,E2 -11087.506} C_VEL
LIN {X 0,Y 397.106,Z 525.828,A -85,B 0,C 180,E1 -11090.729,E2 -11090.729} C_VEL
LIN {X 0,Y 397.131,Z 525.831,A -85,B 0,C 180,E1 -11094.018,E2 -11094.018} C_VEL
LIN {X 0,Y 397.196,Z 525.818,A -85,B 0,C 180,E1 -11097.389,E2 -11097.389} C_VEL
LIN {X 0,Y 397.08,Z 525.831,A -85,B 0,C 180,E1 -11100.882,E2 -11100.882} C_VEL
LIN {X 0,Y 397.126,Z 525.828,A -85,B 0,C 180,E1 -11104.492,E2 -11104.492} C_VEL
LIN {X 0,Y 397.109,Z 525.832,A -85,B 0,C 180,E1 -11108.273,E2 -11108.273} C_VEL
LIN {X 0,Y 397.155,Z 525.828,A -85,B 0,C 180,E1 -11111.992,E2 -11111.992} C_VEL
LIN {X 0,Y 397.111,Z 525.827,A -85,B 0,C 180,E1 -11115.064,E2 -11115.064} C_VEL
LIN {X 0,Y 397.065,Z 525.839,A -85,B 0,C 180,E1 -11118.02,E2 -11118.02} C_VEL
LIN {X 0,Y 397.131,Z 525.825,A -85,B 0,C 180,E1 -11121.137,E2 -11121.137} C_VEL
LIN {X 0,Y 397.116,Z 525.83,A -85,B 0,C 180,E1 -11124.496,E2 -11124.496} C_VEL
LIN {X 0,Y 397.107,Z 525.832,A -85,B 0,C 180,E1 -11127.931,E2 -11127.931} C_VEL
LIN {X 0,Y 397.122,Z 525.826,A -85,B 0,C 180,E1 -11131.456,E2 -11131.456} C_VEL
LIN {X 0,Y 397.147,Z 525.828,A -85,B 0,C 180,E1 -11134.487,E2 -11134.487} C_VEL
LIN {X 0,Y 397.104,Z 525.834,A -85,B 0,C 180,E1 -11138.181,E2 -11138.181} C_VEL
LIN {X 0,Y 397.165,Z 525.821,A -85,B 0,C 180,E1 -11141.426,E2 -11141.426} C_VEL
LIN {X 0,Y 397.173,Z 525.824,A -85,B 0,C 180,E1 -11144.607,E2 -11144.607} C_VEL
LIN {X 0,Y 397.222,Z 525.815,A -85,B 0,C 180,E1 -11147.742,E2 -11147.742} C_VEL
LIN {X 0,Y 397.388,Z 525.796,A -85,B 0,C 180,E1 -11152.04,E2 -11152.04} C_VEL
LIN {X 0,Y 397.25,Z 525.812,A -85,B 0,C 180,E1 -11154.925,E2 -11154.925} C_VEL
LIN {X 0,Y 397.444,Z 525.788,A -85,B 0,C 180,E1 -11157.973,E2 -11157.973} C_VEL
LIN {X 0,Y 397.572,Z 525.772,A -85,B 0,C 180,E1 -11160,E2 -11160} C_VEL
LIN {X 0,Y 397.374,Z 525.796,A -85,B 0,C 180,E1 -11163.041,E2 -11163.041} C_VEL
LIN {X 0,Y 397.366,Z 525.798,A -85,B 0,C 180,E1 -11166.091,E2 -11166.091} C_VEL
LIN {X 0,Y 397.244,Z 525.812,A -85,B 0,C 180,E1 -11169.162,E2 -11169.162} C_VEL
LIN {X 0,Y 397.211,Z 525.818,A -85,B 0,C 180,E1 -11172.258,E2 -11172.258} C_VEL
LIN {X 0,Y 397.171,Z 525.82,A -85,B 0,C 180,E1 -11175.392,E2 -11175.392} C_VEL
LIN {X 0,Y 397.154,Z 525.829,A -85,B 0,C 180,E1 -11178.573,E2 -11178.573} C_VEL
LIN {X 0,Y 397.088,Z 525.83,A -85,B 0,C 180,E1 -11181.819,E2 -11181.819} C_VEL
LIN {X 0,Y 397.145,Z 525.823,A -85,B 0,C 180,E1 -11185.513,E2 -11185.513} C_VEL
LIN {X 0,Y 397.12,Z 525.831,A -85,B 0,C 180,E1 -11188.543,E2 -11188.543} C_VEL
LIN {X 0,Y 397.073,Z 525.833,A -85,B 0,C 180,E1 -11192.072,E2 -11192.072} C_VEL
LIN {X 0,Y 397.114,Z 525.828,A -85,B 0,C 180,E1 -11195.504,E2 -11195.504} C_VEL
LIN {X 0,Y 397.125,Z 525.832,A -85,B 0,C 180,E1 -11198.862,E2 -11198.862} C_VEL
LIN {X 0,Y 397.065,Z 525.834,A -85,B 0,C 180,E1 -11202.267,E2 -11202.267} C_VEL
LIN {X 0,Y 397.087,Z 525.835,A -85,B 0,C 180,E1 -11205.068,E2 -11205.068} C_VEL
LIN {X 0,Y 397.063,Z 525.833,A -85,B 0,C 180,E1 -11208.021,E2 -11208.021} C_VEL
LIN {X 0,Y 397.13,Z 525.829,A -85,B 0,C 180,E1 -11211.138,E2 -11211.138} C_VEL
LIN {X 0,Y 397.116,Z 525.832,A -85,B 0,C 180,E1 -11214.497,E2 -11214.497} C_VEL
LIN {X 0,Y 397.166,Z 525.988,A -85,B 0,C 180,E1 -11216.816,E2 -11216.816} C_VEL
LIN {X 0,Y 399.793,Z 539.048,A -85,B 0,C 180,E1 -11219.937,E2 -11219.937} C_VEL
LIN {X 0,Y 400.675,Z 544.955,A -85,B 0,C 180,E1 -11221.284,E2 -11221.284} C_VEL
LIN {X 0,Y 399.306,Z 562.402,A -85,B 0,C 180,E1 -11225.014,E2 -11225.014} C_VEL
LIN {X 0,Y 397.918,Z 582.866,A -85,B 0,C 180,E1 -11229.315,E2 -11229.315} C_VEL
LIN {X 0,Y 397.078,Z 600.101,A -85,B 0,C 180,E1 -11232.893,E2 -11232.893} C_VEL
LIN {X 0,Y 396.924,Z 604.985,A -85,B 0,C 180,E1 -11233.873,E2 -11233.873} C_VEL
LIN {X 0,Y 397.265,Z 609.413,A -85,B 0,C 180,E1 -11234.034,E2 -11234.034} C_VEL
LIN {X 0,Y 400.307,Z 645.981,A -85,B 0,C 180,E1 -11234.954,E2 -11234.954} C_VEL
LIN {X 0,Y 399.626,Z 688.429,A -85,B 0,C 180,E1 -11235.909,E2 -11235.909} C_VEL
LIN {X 0,Y 399.132,Z 700.388,A -85,B 0,C 180,E1 -11236.379,E2 -11236.379} C_VEL
LIN {X 0,Y 398.504,Z 711.317,A -85,B 0,C 180,E1 -11237.006,E2 -11237.006} C_VEL
LIN {X 0,Y 397.925,Z 721.254,A -85,B 0,C 180,E1 -11237.764,E2 -11237.764} C_VEL
LIN {X 0,Y 397.29,Z 731.565,A -85,B 0,C 180,E1 -11238.78,E2 -11238.78} C_VEL
LIN {X 0,Y 396.89,Z 739.776,A -85,B 0,C 180,E1 -11239.801,E2 -11239.801} C_VEL
LIN {X 0,Y 396.457,Z 748.023,A -85,B 0,C 180,E1 -11241.077,E2 -11241.077} C_VEL
LIN {X 0,Y 396.324,Z 754.595,A -85,B 0,C 180,E1 -11242.357,E2 -11242.357} C_VEL
LIN {X 0,Y 396.353,Z 760.759,A -85,B 0,C 180,E1 -11243.893,E2 -11243.893} C_VEL
LIN {X 0,Y 396.406,Z 765.271,A -85,B 0,C 180,E1 -11245.424,E2 -11245.424} C_VEL
LIN {X 0,Y 396.51,Z 768.408,A -85,B 0,C 180,E1 -11246.952,E2 -11246.952} C_VEL
LIN {X 0,Y 396.532,Z 769.744,A -85,B 0,C 180,E1 -11247.969,E2 -11247.969} C_VEL
LIN {X 0,Y 396.583,Z 770.567,A -85,B 0,C 180,E1 -11248.985,E2 -11248.985} C_VEL
LIN {X 0,Y 396.821,Z 770.838,A -85,B 0,C 180,E1 -11250,E2 -11250} C_VEL
LIN {X 0,Y 396.585,Z 770.534,A -85,B 0,C 180,E1 -11251.015,E2 -11251.015} C_VEL
LIN {X 0,Y 396.53,Z 769.694,A -85,B 0,C 180,E1 -11252.031,E2 -11252.031} C_VEL
LIN {X 0,Y 396.497,Z 768.329,A -85,B 0,C 180,E1 -11253.048,E2 -11253.048} C_VEL
LIN {X 0,Y 396.415,Z 765.212,A -85,B 0,C 180,E1 -11254.576,E2 -11254.576} C_VEL
LIN {X 0,Y 396.312,Z 760.735,A -85,B 0,C 180,E1 -11256.108,E2 -11256.108} C_VEL
LIN {X 0,Y 396.297,Z 754.709,A -85,B 0,C 180,E1 -11257.643,E2 -11257.643} C_VEL
LIN {X 0,Y 396.45,Z 748.345,A -85,B 0,C 180,E1 -11258.923,E2 -11258.923} C_VEL
LIN {X 0,Y 396.834,Z 740.411,A -85,B 0,C 180,E1 -11260.201,E2 -11260.201} C_VEL
LIN {X 0,Y 397.373,Z 731.596,A -85,B 0,C 180,E1 -11261.347,E2 -11261.347} C_VEL
LIN {X 0,Y 398.144,Z 720.458,A -85,B 0,C 180,E1 -11262.488,E2 -11262.488} C_VEL
LIN {X 0,Y 398.945,Z 709.199,A -85,B 0,C 180,E1 -11263.368,E2 -11263.368} C_VEL
LIN {X 0,Y 399.708,Z 697.386,A -85,B 0,C 180,E1 -11264.055,E2 -11264.055} C_VEL
LIN {X 0,Y 400.262,Z 685.516,A -85,B 0,C 180,E1 -11264.54,E2 -11264.54} C_VEL
LIN {X 0,Y 400.657,Z 668.093,A -85,B 0,C 180,E1 -11264.956,E2 -11264.956} C_VEL
LIN {X 0,Y 400.85,Z 642.981,A -85,B 0,C 180,E1 -11265.499,E2 -11265.499} C_VEL
LIN {X 0,Y 398.764,Z 613.518,A -85,B 0,C 180,E1 -11266.263,E2 -11266.263} C_VEL
LIN {X 0,Y 396.89,Z 596.992,A -85,B 0,C 180,E1 -11266.76,E2 -11266.76} C_VEL
LIN {X 0,Y 396.926,Z 595.12,A -85,B 0,C 180,E1 -11267.036,E2 -11267.036} C_VEL
LIN {X 0,Y 397.604,Z 575.787,A -85,B 0,C 180,E1 -11270.973,E2 -11270.973} C_VEL
LIN {X 0,Y 398.563,Z 557.749,A -85,B 0,C 180,E1 -11274.758,E2 -11274.758} C_VEL
LIN {X 0,Y 399.715,Z 541.295,A -85,B 0,C 180,E1 -11278.341,E2 -11278.341} C_VEL
LIN {X 0,Y 399.145,Z 536.206,A -85,B 0,C 180,E1 -11279.538,E2 -11279.538} C_VEL
LIN {X 0,Y 397.183,Z 526.159,A -85,B 0,C 180,E1 -11282.061,E2 -11282.061} C_VEL
LIN {X 0,Y 397.117,Z 525.834,A -85,B 0,C 180,E1 -11282.367,E2 -11282.367} C_VEL
LIN {X 0,Y 397.105,Z 525.833,A -85,B 0,C 180,E1 -11285.734,E2 -11285.734} C_VEL
LIN {X 0,Y 397.11,Z 525.83,A -85,B 0,C 180,E1 -11289.576,E2 -11289.576} C_VEL
LIN {X 0,Y 397.1,Z 525.832,A -85,B 0,C 180,E1 -11293.479,E2 -11293.479} C_VEL
LIN {X 0,Y 397.157,Z 525.826,A -85,B 0,C 180,E1 -11296.511,E2 -11296.511} C_VEL
LIN {X 0,Y 397.117,Z 525.83,A -85,B 0,C 180,E1 -11299.55,E2 -11299.55} C_VEL
LIN {X 0,Y 397.117,Z 525.833,A -85,B 0,C 180,E1 -11302.785,E2 -11302.785} C_VEL
LIN {X 0,Y 397.111,Z 525.831,A -85,B 0,C 180,E1 -11306.282,E2 -11306.282} C_VEL
LIN {X 0,Y 397.081,Z 525.837,A -85,B 0,C 180,E1 -11309.118,E2 -11309.118} C_VEL
LIN {X 0,Y 397.187,Z 525.824,A -85,B 0,C 180,E1 -11312.61,E2 -11312.61} C_VEL
LIN {X 0,Y 397.124,Z 525.827,A -85,B 0,C 180,E1 -11315.982,E2 -11315.982} C_VEL
LIN {X 0,Y 397.13,Z 525.825,A -85,B 0,C 180,E1 -11319.705,E2 -11319.705} C_VEL
LIN {X 0,Y 397.173,Z 525.823,A -85,B 0,C 180,E1 -11322.845,E2 -11322.845} C_VEL
LIN {X 0,Y 397.218,Z 525.819,A -85,B 0,C 180,E1 -11326.679,E2 -11326.679} C_VEL
LIN {X 0,Y 397.221,Z 525.818,A -85,B 0,C 180,E1 -11329.809,E2 -11329.809} C_VEL
LIN {X 0,Y 397.356,Z 525.803,A -85,B 0,C 180,E1 -11332.888,E2 -11332.888} C_VEL
LIN {X 0,Y 397.255,Z 525.816,A -85,B 0,C 180,E1 -11334.925,E2 -11334.925} C_VEL
LIN {X 0,Y 397.443,Z 525.791,A -85,B 0,C 180,E1 -11337.974,E2 -11337.974} C_VEL
LIN {X 0,Y 397.573,Z 525.776,A -85,B 0,C 180,E1 -11340,E2 -11340} C_VEL
LIN {X 0,Y 397.429,Z 526.025,A -85,B 0,C 180,E1 -11342.471,E2 -11342.471} C_VEL
LIN {X 0,Y 397.656,Z 527.056,A -85,B 0,C 180,E1 -11342.628,E2 -11342.628} C_VEL
LIN {X 0,Y 402.729,Z 540.304,A -85,B 0,C 180,E1 -11343.191,E2 -11343.191} C_VEL
LIN {X 0,Y 402.85,Z 562.591,A -85,B 0,C 180,E1 -11343.657,E2 -11343.657} C_VEL
LIN {X 0,Y 402.743,Z 575.384,A -85,B 0,C 180,E1 -11344.121,E2 -11344.121} C_VEL
LIN {X 0,Y 402.542,Z 587.564,A -85,B 0,C 180,E1 -11344.775,E2 -11344.775} C_VEL
LIN {X 0,Y 402.033,Z 599.515,A -85,B 0,C 180,E1 -11345.643,E2 -11345.643} C_VEL
LIN {X 0,Y 401.492,Z 610.336,A -85,B 0,C 180,E1 -11346.66,E2 -11346.66} C_VEL
LIN {X 0,Y 400.847,Z 620.027,A -85,B 0,C 180,E1 -11347.81,E2 -11347.81} C_VEL
LIN {X 0,Y 400.21,Z 628.775,A -85,B 0,C 180,E1 -11349.094,E2 -11349.094} C_VEL
LIN {X 0,Y 399.56,Z 635.988,A -85,B 0,C 180,E1 -11350.387,E2 -11350.387} C_VEL
LIN {X 0,Y 398.944,Z 642.943,A -85,B 0,C 180,E1 -11351.947,E2 -11351.947} C_VEL
LIN {X 0,Y 398.313,Z 649.088,A -85,B 0,C 180,E1 -11353.741,E2 -11353.741} C_VEL
LIN {X 0,Y 397.849,Z 653.226,A -85,B 0,C 180,E1 -11355.366,E2 -11355.366} C_VEL
LIN {X 0,Y 397.458,Z 656.501,A -85,B 0,C 180,E1 -11357.288,E2 -11357.288} C_VEL
LIN {X 0,Y 397.283,Z 657.839,A -85,B 0,C 180,E1 -11358.568,E2 -11358.568} C_VEL
LIN {X 0,Y 397.123,Z 658.564,A -85,B 0,C 180,E1 -11360.293,E2 -11360.293} C_VEL
LIN {X 0,Y 397.055,Z 658.221,A -85,B 0,C 180,E1 -11361.821,E2 -11361.821} C_VEL
LIN {X 0,Y 397.08,Z 657.305,A -85,B 0,C 180,E1 -11363.025,E2 -11363.025} C_VEL
LIN {X 0,Y 397.114,Z 656.091,A -85,B 0,C 180,E1 -11364.02,E2 -11364.02} C_VEL
LIN {X 0,Y 397.333,Z 653.368,A -85,B 0,C 180,E1 -11365.57,E2 -11365.57} C_VEL
LIN {X 0,Y 397.592,Z 648.893,A -85,B 0,C 180,E1 -11367.361,E2 -11367.361} C_VEL
LIN {X 0,Y 397.96,Z 643.206,A -85,B 0,C 180,E1 -11369.056,E2 -11369.056} C_VEL
LIN {X 0,Y 398.441,Z 635.712,A -85,B 0,C 180,E1 -11370.766,E2 -11370.766} C_VEL
LIN {X 0,Y 399.032,Z 627.297,A -85,B 0,C 180,E1 -11372.287,E2 -11372.287} C_VEL
LIN {X 0,Y 399.565,Z 617.882,A -85,B 0,C 180,E1 -11373.646,E2 -11373.646} C_VEL
LIN {X 0,Y 400.134,Z 606.94,A -85,B 0,C 180,E1 -11374.916,E2 -11374.916} C_VEL
LIN {X 0,Y 400.683,Z 595.883,A -85,B 0,C 180,E1 -11375.923,E2 -11375.923} C_VEL
LIN {X 0,Y 401.076,Z 583.555,A -85,B 0,C 180,E1 -11376.803,E2 -11376.803} C_VEL
LIN {X 0,Y 401.349,Z 570.915,A -85,B 0,C 180,E1 -11377.462,E2 -11377.462} C_VEL
LIN {X 0,Y 401.439,Z 557.52,A -85,B 0,C 180,E1 -11377.938,E2 -11377.938} C_VEL
LIN {X 0,Y 401.38,Z 539.33,A -85,B 0,C 180,E1 -11378.321,E2 -11378.321} C_VEL
LIN {X 0,Y 397.324,Z 526.733,A -85,B 0,C 180,E1 -11378.742,E2 -11378.742} C_VEL
LIN {X 0,Y 397.172,Z 525.917,A -85,B 0,C 180,E1 -11378.926,E2 -11378.926} C_VEL
LIN {X 0,Y 397.068,Z 525.836,A -85,B 0,C 180,E1 -11382.268,E2 -11382.268} C_VEL
LIN {X 0,Y 397.115,Z 525.83,A -85,B 0,C 180,E1 -11385.065,E2 -11385.065} C_VEL
LIN {X 0,Y 397.154,Z 525.823,A -85,B 0,C 180,E1 -11388.008,E2 -11388.008} C_VEL
LIN {X 0,Y 397.109,Z 525.831,A -85,B 0,C 180,E1 -11391.727,E2 -11391.727} C_VEL
LIN {X 0,Y 397.126,Z 525.832,A -85,B 0,C 180,E1 -11395.508,E2 -11395.508} C_VEL
LIN {X 0,Y 397.079,Z 525.834,A -85,B 0,C 180,E1 -11399.119,E2 -11399.119} C_VEL
LIN {X 0,Y 397.196,Z 525.817,A -85,B 0,C 180,E1 -11402.611,E2 -11402.611} C_VEL
LIN {X 0,Y 397.136,Z 525.827,A -85,B 0,C 180,E1 -11405.983,E2 -11405.983} C_VEL
LIN {X 0,Y 397.147,Z 525.829,A -85,B 0,C 180,E1 -11409.703,E2 -11409.703} C_VEL
LIN {X 0,Y 397.185,Z 525.819,A -85,B 0,C 180,E1 -11412.846,E2 -11412.846} C_VEL
LIN {X 0,Y 397.233,Z 525.812,A -85,B 0,C 180,E1 -11416.703,E2 -11416.703} C_VEL
LIN {X 0,Y 397.221,Z 525.819,A -85,B 0,C 180,E1 -11419.809,E2 -11419.809} C_VEL
LIN {X 0,Y 397.322,Z 525.801,A -85,B 0,C 180,E1 -11422.888,E2 -11422.888} C_VEL
LIN {X 0,Y 397.251,Z 525.81,A -85,B 0,C 180,E1 -11424.925,E2 -11424.925} C_VEL
LIN {X 0,Y 397.454,Z 525.789,A -85,B 0,C 180,E1 -11427.973,E2 -11427.973} C_VEL
LIN {X 0,Y 397.584,Z 525.773,A -85,B 0,C 180,E1 -11430,E2 -11430} C_VEL
LIN {X 0,Y 397.38,Z 525.794,A -85,B 0,C 180,E1 -11433.041,E2 -11433.041} C_VEL
LIN {X 0,Y 397.349,Z 525.801,A -85,B 0,C 180,E1 -11436.092,E2 -11436.092} C_VEL
LIN {X 0,Y 397.311,Z 525.809,A -85,B 0,C 180,E1 -11437.889,E2 -11437.889} C_VEL
LIN {X 0,Y 396.562,Z 525.897,A -85,B 0,C 180,E1 -11438.734,E2 -11438.734} C_VEL
LIN {X 0,Y 393.635,Z 526.264,A -85,B 0,C 180,E1 -11440.107,E2 -11440.107} C_VEL
LIN {X 0,Y 391.224,Z 526.562,A -85,B 0,C 180,E1 -11441.216,E2 -11441.216} C_VEL
LIN {X 0,Y 390.229,Z 526.689,A -85,B 0,C 180,E1 -11442.075,E2 -11442.075} C_VEL
LIN {X 0,Y 390.166,Z 526.693,A -85,B 0,C 180,E1 -11442.365,E2 -11442.365} C_VEL
LIN {X 0,Y 390.143,Z 526.7,A -85,B 0,C 180,E1 -11445.676,E2 -11445.676} C_VEL
LIN {X 0,Y 390.109,Z 526.7,A -85,B 0,C 180,E1 -11448.921,E2 -11448.921} C_VEL
LIN {X 0,Y 390.04,Z 526.712,A -85,B 0,C 180,E1 -11452.234,E2 -11452.234} C_VEL
LIN {X 0,Y 390.121,Z 526.703,A -85,B 0,C 180,E1 -11455.743,E2 -11455.743} C_VEL
LIN {X 0,Y 390.06,Z 526.706,A -85,B 0,C 180,E1 -11459.109,E2 -11459.109} C_VEL
LIN {X 0,Y 390.044,Z 526.708,A -85,B 0,C 180,E1 -11462.721,E2 -11462.721} C_VEL
LIN {X 0,Y 390.058,Z 526.711,A -85,B 0,C 180,E1 -11465.825,E2 -11465.825} C_VEL
LIN {X 0,Y 390.074,Z 526.704,A -85,B 0,C 180,E1 -11469.218,E2 -11469.218} C_VEL
LIN {X 0,Y 390.12,Z 526.702,A -85,B 0,C 180,E1 -11472.386,E2 -11472.386} C_VEL
LIN {X 0,Y 390.061,Z 526.706,A -85,B 0,C 180,E1 -11475.356,E2 -11475.356} C_VEL
LIN {X 0,Y 390.029,Z 526.716,A -85,B 0,C 180,E1 -11478.186,E2 -11478.186} C_VEL
LIN {X 0,Y 390.09,Z 526.702,A -85,B 0,C 180,E1 -11480.907,E2 -11480.907} C_VEL
LIN {X 0,Y 390.082,Z 526.704,A -85,B 0,C 180,E1 -11484.792,E2 -11484.792} C_VEL
LIN {X 0,Y 390.045,Z 526.711,A -85,B 0,C 180,E1 -11488.497,E2 -11488.497} C_VEL
LIN {X 0,Y 390.113,Z 526.704,A -85,B 0,C 180,E1 -11492.069,E2 -11492.069} C_VEL
LIN {X 0,Y 390.074,Z 526.704,A -85,B 0,C 180,E1 -11495.518,E2 -11495.518} C_VEL
LIN {X 0,Y 390.066,Z 526.706,A -85,B 0,C 180,E1 -11498.878,E2 -11498.878} C_VEL
LIN {X 0,Y 390.124,Z 526.703,A -85,B 0,C 180,E1 -11502.166,E2 -11502.166} C_VEL
LIN {X 0,Y 390.14,Z 526.696,A -85,B 0,C 180,E1 -11505.392,E2 -11505.392} C_VEL
LIN {X 0,Y 390.151,Z 526.699,A -85,B 0,C 180,E1 -11508.571,E2 -11508.571} C_VEL
LIN {X 0,Y 390.337,Z 526.674,A -85,B 0,C 180,E1 -11511.993,E2 -11511.993} C_VEL
LIN {X 0,Y 390.222,Z 526.688,A -85,B 0,C 180,E1 -11514.833,E2 -11514.833} C_VEL
LIN {X 0,Y 390.413,Z 526.663,A -85,B 0,C 180,E1 -11517.936,E2 -11517.936} C_VEL
LIN {X 0,Y 390.542,Z 526.648,A -85,B 0,C 180,E1 -11520,E2 -11520} C_VEL
LIN {X 0,Y 390.308,Z 526.676,A -85,B 0,C 180,E1 -11523.096,E2 -11523.096} C_VEL
LIN {X 0,Y 390.319,Z 526.677,A -85,B 0,C 180,E1 -11526.202,E2 -11526.202} C_VEL
LIN {X 0,Y 390.197,Z 526.689,A -85,B 0,C 180,E1 -11529.329,E2 -11529.329} C_VEL
LIN {X 0,Y 390.186,Z 526.69,A -85,B 0,C 180,E1 -11533.438,E2 -11533.438} C_VEL
LIN {X 0,Y 390.141,Z 526.696,A -85,B 0,C 180,E1 -11537.308,E2 -11537.308} C_VEL
LIN {X 0,Y 390.079,Z 526.708,A -85,B 0,C 180,E1 -11540.47,E2 -11540.47} C_VEL
LIN {X 0,Y 390.07,Z 526.709,A -85,B 0,C 180,E1 -11544.481,E2 -11544.481} C_VEL
LIN {X 0,Y 390.109,Z 526.7,A -85,B 0,C 180,E1 -11548.025,E2 -11548.025} C_VEL
LIN {X 0,Y 390.02,Z 526.711,A -85,B 0,C 180,E1 -11551.504,E2 -11551.504} C_VEL
LIN {X 0,Y 390.079,Z 526.706,A -85,B 0,C 180,E1 -11555.207,E2 -11555.207} C_VEL
LIN {X 0,Y 390.085,Z 526.706,A -85,B 0,C 180,E1 -11559.093,E2 -11559.093} C_VEL
LIN {X 0,Y 390.039,Z 526.711,A -85,B 0,C 180,E1 -11562.375,E2 -11562.375} C_VEL
LIN {X 0,Y 390.043,Z 526.71,A -85,B 0,C 180,E1 -11565.355,E2 -11565.355} C_VEL
LIN {X 0,Y 390.028,Z 526.71,A -85,B 0,C 180,E1 -11568.187,E2 -11568.187} C_VEL
LIN {X 0,Y 390.089,Z 526.71,A -85,B 0,C 180,E1 -11570.908,E2 -11570.908} C_VEL
LIN {X 0,Y 390.083,Z 526.71,A -85,B 0,C 180,E1 -11574.794,E2 -11574.794} C_VEL
LIN {X 0,Y 390.129,Z 526.842,A -85,B 0,C 180,E1 -11576.595,E2 -11576.595} C_VEL
LIN {X 0,Y 392.879,Z 540.566,A -85,B 0,C 180,E1 -11579.943,E2 -11579.943} C_VEL
LIN {X 0,Y 393.675,Z 545.899,A -85,B 0,C 180,E1 -11581.184,E2 -11581.184} C_VEL
LIN {X 0,Y 392.294,Z 562.557,A -85,B 0,C 180,E1 -11584.819,E2 -11584.819} C_VEL
LIN {X 0,Y 390.963,Z 581.683,A -85,B 0,C 180,E1 -11588.93,E2 -11588.93} C_VEL
LIN {X 0,Y 390.012,Z 599.697,A -85,B 0,C 180,E1 -11592.757,E2 -11592.757} C_VEL
LIN {X 0,Y 389.889,Z 603.872,A -85,B 0,C 180,E1 -11593.608,E2 -11593.608} C_VEL
LIN {X 0,Y 390.725,Z 614.121,A -85,B 0,C 180,E1 -11593.912,E2 -11593.912} C_VEL
LIN {X 0,Y 393.354,Z 646.541,A -85,B 0,C 180,E1 -11594.754,E2 -11594.754} C_VEL
LIN {X 0,Y 392.705,Z 687.002,A -85,B 0,C 180,E1 -11595.689,E2 -11595.689} C_VEL
LIN {X 0,Y 392.227,Z 698.425,A -85,B 0,C 180,E1 -11596.134,E2 -11596.134} C_VEL
LIN {X 0,Y 391.536,Z 709.557,A -85,B 0,C 180,E1 -11596.77,E2 -11596.77} C_VEL
LIN {X 0,Y 390.972,Z 719.681,A -85,B 0,C 180,E1 -11597.543,E2 -11597.543} C_VEL
LIN {X 0,Y 390.332,Z 728.898,A -85,B 0,C 180,E1 -11598.445,E2 -11598.445} C_VEL
LIN {X 0,Y 389.815,Z 738.393,A -85,B 0,C 180,E1 -11599.613,E2 -11599.613} C_VEL
LIN {X 0,Y 389.414,Z 746.711,A -85,B 0,C 180,E1 -11600.914,E2 -11600.914} C_VEL
LIN {X 0,Y 389.29,Z 753.364,A -85,B 0,C 180,E1 -11602.218,E2 -11602.218} C_VEL
LIN {X 0,Y 389.297,Z 759.572,A -85,B 0,C 180,E1 -11603.782,E2 -11603.782} C_VEL
LIN {X 0,Y 389.344,Z 764.142,A -85,B 0,C 180,E1 -11605.341,E2 -11605.341} C_VEL
LIN {X 0,Y 389.471,Z 767.317,A -85,B 0,C 180,E1 -11606.897,E2 -11606.897} C_VEL
LIN {X 0,Y 389.497,Z 768.685,A -85,B 0,C 180,E1 -11607.932,E2 -11607.932} C_VEL
LIN {X 0,Y 389.553,Z 769.527,A -85,B 0,C 180,E1 -11608.966,E2 -11608.966} C_VEL
LIN {X 0,Y 389.794,Z 769.819,A -85,B 0,C 180,E1 -11610,E2 -11610} C_VEL
LIN {X 0,Y 389.549,Z 769.533,A -85,B 0,C 180,E1 -11611.034,E2 -11611.034} C_VEL
LIN {X 0,Y 389.485,Z 768.703,A -85,B 0,C 180,E1 -11612.068,E2 -11612.068} C_VEL
LIN {X 0,Y 389.446,Z 767.358,A -85,B 0,C 180,E1 -11613.103,E2 -11613.103} C_VEL
LIN {X 0,Y 389.347,Z 764.25,A -85,B 0,C 180,E1 -11614.659,E2 -11614.659} C_VEL
LIN {X 0,Y 389.223,Z 759.798,A -85,B 0,C 180,E1 -11616.219,E2 -11616.219} C_VEL
LIN {X 0,Y 389.221,Z 753.787,A -85,B 0,C 180,E1 -11617.783,E2 -11617.783} C_VEL
LIN {X 0,Y 389.388,Z 747.47,A -85,B 0,C 180,E1 -11619.086,E2 -11619.086} C_VEL
LIN {X 0,Y 389.776,Z 739.613,A -85,B 0,C 180,E1 -11620.387,E2 -11620.387} C_VEL
LIN {X 0,Y 390.309,Z 730.904,A -85,B 0,C 180,E1 -11621.555,E2 -11621.555} C_VEL
LIN {X 0,Y 391.093,Z 721.26,A -85,B 0,C 180,E1 -11622.585,E2 -11622.585} C_VEL
LIN {X 0,Y 391.877,Z 710.658,A -85,B 0,C 180,E1 -11623.482,E2 -11623.482} C_VEL
LIN {X 0,Y 392.749,Z 698.618,A -85,B 0,C 180,E1 -11624.243,E2 -11624.243} C_VEL
LIN {X 0,Y 393.416,Z 685.856,A -85,B 0,C 180,E1 -11624.808,E2 -11624.808} C_VEL
LIN {X 0,Y 393.777,Z 673.693,A -85,B 0,C 180,E1 -11625.144,E2 -11625.144} C_VEL
LIN {X 0,Y 394.08,Z 643.501,A -85,B 0,C 180,E1 -11625.809,E2 -11625.809} C_VEL
LIN {X 0,Y 392.2,Z 615.188,A -85,B 0,C 180,E1 -11626.568,E2 -11626.568} C_VEL
LIN {X 0,Y 389.892,Z 595.299,A -85,B 0,C 180,E1 -11627.187,E2 -11627.187} C_VEL
LIN {X 0,Y 389.896,Z 593.575,A -85,B 0,C 180,E1 -11627.437,E2 -11627.437} C_VEL
LIN {X 0,Y 390.689,Z 573.447,A -85,B 0,C 180,E1 -11631.639,E2 -11631.639} C_VEL
LIN {X 0,Y 391.626,Z 556.814,A -85,B 0,C 180,E1 -11635.227,E2 -11635.227} C_VEL
LIN {X 0,Y 392.713,Z 542.999,A -85,B 0,C 180,E1 -11638.309,E2 -11638.309} C_VEL
LIN {X 0,Y 392.503,Z 539.213,A -85,B 0,C 180,E1 -11639.204,E2 -11639.204} C_VEL
LIN {X 0,Y 390.238,Z 527.576,A -85,B 0,C 180,E1 -11642.173,E2 -11642.173} C_VEL
LIN {X 0,Y 390.084,Z 526.716,A -85,B 0,C 180,E1 -11642.549,E2 -11642.549} C_VEL
LIN {X 0,Y 390.053,Z 526.711,A -85,B 0,C 180,E1 -11645.825,E2 -11645.825} C_VEL
LIN {X 0,Y 390.067,Z 526.711,A -85,B 0,C 180,E1 -11649.218,E2 -11649.218} C_VEL
LIN {X 0,Y 390.039,Z 526.71,A -85,B 0,C 180,E1 -11652.374,E2 -11652.374} C_VEL
LIN {X 0,Y 390.098,Z 526.703,A -85,B 0,C 180,E1 -11656.106,E2 -11656.106} C_VEL
LIN {X 0,Y 390.076,Z 526.71,A -85,B 0,C 180,E1 -11659.174,E2 -11659.174} C_VEL
LIN {X 0,Y 390.053,Z 526.71,A -85,B 0,C 180,E1 -11662.445,E2 -11662.445} C_VEL
LIN {X 0,Y 390.06,Z 526.708,A -85,B 0,C 180,E1 -11666.045,E2 -11666.045} C_VEL
LIN {X 0,Y 390.041,Z 526.71,A -85,B 0,C 180,E1 -11668.498,E2 -11668.498} C_VEL
LIN {X 0,Y 390.109,Z 526.702,A -85,B 0,C 180,E1 -11672.07,E2 -11672.07} C_VEL
LIN {X 0,Y 390.071,Z 526.707,A -85,B 0,C 180,E1 -11675.519,E2 -11675.519} C_VEL
LIN {X 0,Y 390.054,Z 526.71,A -85,B 0,C 180,E1 -11678.878,E2 -11678.878} C_VEL
LIN {X 0,Y 390.119,Z 526.699,A -85,B 0,C 180,E1 -11682.167,E2 -11682.167} C_VEL
LIN {X 0,Y 390.138,Z 526.701,A -85,B 0,C 180,E1 -11685.393,E2 -11685.393} C_VEL
LIN {X 0,Y 390.152,Z 526.701,A -85,B 0,C 180,E1 -11688.572,E2 -11688.572} C_VEL
LIN {X 0,Y 390.335,Z 526.677,A -85,B 0,C 180,E1 -11691.993,E2 -11691.993} C_VEL
LIN {X 0,Y 390.227,Z 526.691,A -85,B 0,C 180,E1 -11694.834,E2 -11694.834} C_VEL
LIN {X 0,Y 390.412,Z 526.667,A -85,B 0,C 180,E1 -11697.937,E2 -11697.937} C_VEL
LIN {X 0,Y 390.543,Z 526.652,A -85,B 0,C 180,E1 -11700,E2 -11700} C_VEL
LIN {X 0,Y 390.422,Z 526.882,A -85,B 0,C 180,E1 -11702.064,E2 -11702.064} C_VEL
LIN {X 0,Y 390.705,Z 528.049,A -85,B 0,C 180,E1 -11702.239,E2 -11702.239} C_VEL
LIN {X 0,Y 396.064,Z 541.711,A -85,B 0,C 180,E1 -11702.842,E2 -11702.842} C_VEL
LIN {X 0,Y 396.21,Z 565.419,A -85,B 0,C 180,E1 -11703.376,E2 -11703.376} C_VEL
LIN {X 0,Y 396.092,Z 577.206,A -85,B 0,C 180,E1 -11703.826,E2 -11703.826} C_VEL
LIN {X 0,Y 395.897,Z 588.764,A -85,B 0,C 180,E1 -11704.464,E2 -11704.464} C_VEL
LIN {X 0,Y 395.413,Z 599.57,A -85,B 0,C 180,E1 -11705.25,E2 -11705.25} C_VEL
LIN {X 0,Y 394.811,Z 611.032,A -85,B 0,C 180,E1 -11706.326,E2 -11706.326} C_VEL
LIN {X 0,Y 394.181,Z 620.337,A -85,B 0,C 180,E1 -11707.427,E2 -11707.427} C_VEL
LIN {X 0,Y 393.46,Z 629.235,A -85,B 0,C 180,E1 -11708.733,E2 -11708.733} C_VEL
LIN {X 0,Y 392.714,Z 637.212,A -85,B 0,C 180,E1 -11710.181,E2 -11710.181} C_VEL
LIN {X 0,Y 392.1,Z 643.617,A -85,B 0,C 180,E1 -11711.634,E2 -11711.634} C_VEL
LIN {X 0,Y 391.617,Z 648.331,A -85,B 0,C 180,E1 -11712.964,E2 -11712.964} C_VEL
LIN {X 0,Y 391.099,Z 652.819,A -85,B 0,C 180,E1 -11714.571,E2 -11714.571} C_VEL
LIN {X 0,Y 390.797,Z 655.132,A -85,B 0,C 180,E1 -11715.65,E2 -11715.65} C_VEL
LIN {X 0,Y 390.436,Z 657.908,A -85,B 0,C 180,E1 -11717.447,E2 -11717.447} C_VEL
LIN {X 0,Y 390.234,Z 659.18,A -85,B 0,C 180,E1 -11718.916,E2 -11718.916} C_VEL
LIN {X 0,Y 390.094,Z 659.616,A -85,B 0,C 180,E1 -11720.476,E2 -11720.476} C_VEL
LIN {X 0,Y 390.042,Z 658.99,A -85,B 0,C 180,E1 -11722.234,E2 -11722.234} C_VEL
LIN {X 0,Y 390.066,Z 657.943,A -85,B 0,C 180,E1 -11723.353,E2 -11723.353} C_VEL
LIN {X 0,Y 390.221,Z 655.44,A -85,B 0,C 180,E1 -11725.04,E2 -11725.04} C_VEL
LIN {X 0,Y 390.487,Z 651.714,A -85,B 0,C 180,E1 -11726.741,E2 -11726.741} C_VEL
LIN {X 0,Y 390.808,Z 646.244,A -85,B 0,C 180,E1 -11728.562,E2 -11728.562} C_VEL
LIN {X 0,Y 391.229,Z 639.807,A -85,B 0,C 180,E1 -11730.198,E2 -11730.198} C_VEL
LIN {X 0,Y 391.74,Z 632.661,A -85,B 0,C 180,E1 -11731.653,E2 -11731.653} C_VEL
LIN {X 0,Y 392.286,Z 623.7,A -85,B 0,C 180,E1 -11733.122,E2 -11733.122} C_VEL
LIN {X 0,Y 392.928,Z 613.869,A -85,B 0,C 180,E1 -11734.416,E2 -11734.416} C_VEL
LIN {X 0,Y 393.396,Z 603.804,A -85,B 0,C 180,E1 -11735.494,E2 -11735.494} C_VEL
LIN {X 0,Y 393.927,Z 592.242,A -85,B 0,C 180,E1 -11736.468,E2 -11736.468} C_VEL
LIN {X 0,Y 394.282,Z 581.078,A -85,B 0,C 180,E1 -11737.202,E2 -11737.202} C_VEL
LIN {X 0,Y 394.514,Z 568.198,A -85,B 0,C 180,E1 -11737.826,E2 -11737.826} C_VEL
LIN {X 0,Y 394.551,Z 554.753,A -85,B 0,C 180,E1 -11738.243,E2 -11738.243} C_VEL
LIN {X 0,Y 394.519,Z 540.692,A -85,B 0,C 180,E1 -11738.539,E2 -11738.539} C_VEL
LIN {X 0,Y 390.288,Z 527.679,A -85,B 0,C 180,E1 -11738.978,E2 -11738.978} C_VEL
LIN {X 0,Y 390.106,Z 526.788,A -85,B 0,C 180,E1 -11739.181,E2 -11739.181} C_VEL
LIN {X 0,Y 390.042,Z 526.711,A -85,B 0,C 180,E1 -11742.376,E2 -11742.376} C_VEL
LIN {X 0,Y 390.1,Z 526.701,A -85,B 0,C 180,E1 -11746.108,E2 -11746.108} C_VEL
LIN {X 0,Y 390.081,Z 526.708,A -85,B 0,C 180,E1 -11749.175,E2 -11749.175} C_VEL
LIN {X 0,Y 390.046,Z 526.707,A -85,B 0,C 180,E1 -11752.45,E2 -11752.45} C_VEL
LIN {X 0,Y 390.068,Z 526.706,A -85,B 0,C 180,E1 -11756.046,E2 -11756.046} C_VEL
LIN {X 0,Y 390.048,Z 526.71,A -85,B 0,C 180,E1 -11759.87,E2 -11759.87} C_VEL
LIN {X 0,Y 390.115,Z 526.703,A -85,B 0,C 180,E1 -11763.233,E2 -11763.233} C_VEL
LIN {X 0,Y 390.109,Z 526.7,A -85,B 0,C 180,E1 -11766.751,E2 -11766.751} C_VEL
LIN {X 0,Y 390.109,Z 526.702,A -85,B 0,C 180,E1 -11769.984,E2 -11769.984} C_VEL
LIN {X 0,Y 390.141,Z 526.699,A -85,B 0,C 180,E1 -11773.249,E2 -11773.249} C_VEL
LIN {X 0,Y 390.198,Z 526.688,A -85,B 0,C 180,E1 -11776.562,E2 -11776.562} C_VEL
LIN {X 0,Y 390.208,Z 526.687,A -85,B 0,C 180,E1 -11780.672,E2 -11780.672} C_VEL
LIN {X 0,Y 390.303,Z 526.681,A -85,B 0,C 180,E1 -11783.798,E2 -11783.798} C_VEL
LIN {X 0,Y 390.422,Z 526.665,A -85,B 0,C 180,E1 -11787.937,E2 -11787.937} C_VEL
LIN {X 0,Y 390.553,Z 526.648,A -85,B 0,C 180,E1 -11790,E2 -11790} C_VEL
LIN {X 0,Y 390.314,Z 526.675,A -85,B 0,C 180,E1 -11793.097,E2 -11793.097} C_VEL
LIN {X 0,Y 390.303,Z 526.678,A -85,B 0,C 180,E1 -11796.202,E2 -11796.202} C_VEL
LIN {X 0,Y 390.198,Z 526.69,A -85,B 0,C 180,E1 -11799.329,E2 -11799.329} C_VEL
LIN {X 0,Y 390.166,Z 526.693,A -85,B 0,C 180,E1 -11802.365,E2 -11802.365} C_VEL
LIN {X 0,Y 389.532,Z 526.774,A -85,B 0,C 180,E1 -11803.227,E2 -11803.227} C_VEL
LIN {X 0,Y 386.64,Z 527.135,A -85,B 0,C 180,E1 -11804.625,E2 -11804.625} C_VEL
LIN {X 0,Y 384.186,Z 527.443,A -85,B 0,C 180,E1 -11805.756,E2 -11805.756} C_VEL
LIN {X 0,Y 383.163,Z 527.566,A -85,B 0,C 180,E1 -11806.632,E2 -11806.632} C_VEL
LIN {X 0,Y 383.098,Z 527.573,A -85,B 0,C 180,E1 -11806.928,E2 -11806.928} C_VEL
LIN {X 0,Y 383.032,Z 527.582,A -85,B 0,C 180,E1 -11810.646,E2 -11810.646} C_VEL
LIN {X 0,Y 383.025,Z 527.588,A -85,B 0,C 180,E1 -11813.807,E2 -11813.807} C_VEL
LIN {X 0,Y 383.082,Z 527.58,A -85,B 0,C 180,E1 -11816.123,E2 -11816.123} C_VEL
LIN {X 0,Y 382.994,Z 527.59,A -85,B 0,C 180,E1 -11819.699,E2 -11819.699} C_VEL
LIN {X 0,Y 383.013,Z 527.585,A -85,B 0,C 180,E1 -11823.399,E2 -11823.399} C_VEL
LIN {X 0,Y 383.034,Z 527.587,A -85,B 0,C 180,E1 -11826.164,E2 -11826.164} C_VEL
LIN {X 0,Y 383.02,Z 527.588,A -85,B 0,C 180,E1 -11829.956,E2 -11829.956} C_VEL
LIN {X 0,Y 383.064,Z 527.578,A -85,B 0,C 180,E1 -11832.787,E2 -11832.787} C_VEL
LIN {X 0,Y 383.006,Z 527.588,A -85,B 0,C 180,E1 -11835.79,E2 -11835.79} C_VEL
LIN {X 0,Y 382.986,Z 527.588,A -85,B 0,C 180,E1 -11838.795,E2 -11838.795} C_VEL
LIN {X 0,Y 382.999,Z 527.592,A -85,B 0,C 180,E1 -11842.095,E2 -11842.095} C_VEL
LIN {X 0,Y 383.015,Z 527.583,A -85,B 0,C 180,E1 -11845.331,E2 -11845.331} C_VEL
LIN {X 0,Y 383.033,Z 527.584,A -85,B 0,C 180,E1 -11847.852,E2 -11847.852} C_VEL
LIN {X 0,Y 383.06,Z 527.579,A -85,B 0,C 180,E1 -11851.719,E2 -11851.719} C_VEL
LIN {X 0,Y 383.047,Z 527.58,A -85,B 0,C 180,E1 -11855.039,E2 -11855.039} C_VEL
LIN {X 0,Y 382.999,Z 527.591,A -85,B 0,C 180,E1 -11858.469,E2 -11858.469} C_VEL
LIN {X 0,Y 383.087,Z 527.576,A -85,B 0,C 180,E1 -11861.827,E2 -11861.827} C_VEL
LIN {X 0,Y 383.105,Z 527.573,A -85,B 0,C 180,E1 -11865.118,E2 -11865.118} C_VEL
LIN {X 0,Y 383.1,Z 527.58,A -85,B 0,C 180,E1 -11868.358,E2 -11868.358} C_VEL
LIN {X 0,Y 383.297,Z 527.55,A -85,B 0,C 180,E1 -11871.932,E2 -11871.932} C_VEL
LIN {X 0,Y 383.194,Z 527.565,A -85,B 0,C 180,E1 -11874.738,E2 -11874.738} C_VEL
LIN {X 0,Y 383.38,Z 527.539,A -85,B 0,C 180,E1 -11877.898,E2 -11877.898} C_VEL
LIN {X 0,Y 383.511,Z 527.523,A -85,B 0,C 180,E1 -11880,E2 -11880} C_VEL
LIN {X 0,Y 383.245,Z 527.556,A -85,B 0,C 180,E1 -11883.153,E2 -11883.153} C_VEL
LIN {X 0,Y 383.275,Z 527.555,A -85,B 0,C 180,E1 -11886.316,E2 -11886.316} C_VEL
LIN {X 0,Y 383.143,Z 527.567,A -85,B 0,C 180,E1 -11889.502,E2 -11889.502} C_VEL
LIN {X 0,Y 383.117,Z 527.571,A -85,B 0,C 180,E1 -11893.536,E2 -11893.536} C_VEL
LIN {X 0,Y 383.087,Z 527.575,A -85,B 0,C 180,E1 -11897.454,E2 -11897.454} C_VEL
LIN {X 0,Y 383.021,Z 527.59,A -85,B 0,C 180,E1 -11900.647,E2 -11900.647} C_VEL
LIN {X 0,Y 383.018,Z 527.583,A -85,B 0,C 180,E1 -11903.808,E2 -11903.808} C_VEL
LIN {X 0,Y 383.073,Z 527.577,A -85,B 0,C 180,E1 -11906.124,E2 -11906.124} C_VEL
LIN {X 0,Y 383.043,Z 527.584,A -85,B 0,C 180,E1 -11908.492,E2 -11908.492} C_VEL
LIN {X 0,Y 383.004,Z 527.586,A -85,B 0,C 180,E1 -11912.15,E2 -11912.15} C_VEL
LIN {X 0,Y 383.012,Z 527.59,A -85,B 0,C 180,E1 -11914.668,E2 -11914.668} C_VEL
LIN {X 0,Y 382.995,Z 527.586,A -85,B 0,C 180,E1 -11917.904,E2 -11917.904} C_VEL
LIN {X 0,Y 382.978,Z 527.59,A -85,B 0,C 180,E1 -11921.348,E2 -11921.348} C_VEL
LIN {X 0,Y 382.994,Z 527.587,A -85,B 0,C 180,E1 -11924.304,E2 -11924.304} C_VEL
LIN {X 0,Y 383.005,Z 527.588,A -85,B 0,C 180,E1 -11927.241,E2 -11927.241} C_VEL
LIN {X 0,Y 383.013,Z 527.586,A -85,B 0,C 180,E1 -11930.414,E2 -11930.414} C_VEL
LIN {X 0,Y 383.023,Z 527.586,A -85,B 0,C 180,E1 -11934.045,E2 -11934.045} C_VEL
LIN {X 0,Y 383.102,Z 527.714,A -85,B 0,C 180,E1 -11936.377,E2 -11936.377} C_VEL
LIN {X 0,Y 385.962,Z 542.053,A -85,B 0,C 180,E1 -11939.951,E2 -11939.951} C_VEL
LIN {X 0,Y 386.629,Z 547.368,A -85,B 0,C 180,E1 -11941.204,E2 -11941.204} C_VEL
LIN {X 0,Y 385.188,Z 563.952,A -85,B 0,C 180,E1 -11944.9,E2 -11944.9} C_VEL
LIN {X 0,Y 383.836,Z 582.79,A -85,B 0,C 180,E1 -11949.035,E2 -11949.035} C_VEL
LIN {X 0,Y 382.859,Z 601.963,A -85,B 0,C 180,E1 -11953.195,E2 -11953.195} C_VEL
LIN {X 0,Y 382.845,Z 603.244,A -85,B 0,C 180,E1 -11953.366,E2 -11953.366} C_VEL
LIN {X 0,Y 386.42,Z 647.09,A -85,B 0,C 180,E1 -11954.548,E2 -11954.548} C_VEL
LIN {X 0,Y 385.716,Z 686.562,A -85,B 0,C 180,E1 -11955.491,E2 -11955.491} C_VEL
LIN {X 0,Y 385.262,Z 697.754,A -85,B 0,C 180,E1 -11955.946,E2 -11955.946} C_VEL
LIN {X 0,Y 384.479,Z 709.726,A -85,B 0,C 180,E1 -11956.657,E2 -11956.657} C_VEL
LIN {X 0,Y 383.916,Z 719.536,A -85,B 0,C 180,E1 -11957.445,E2 -11957.445} C_VEL
LIN {X 0,Y 383.269,Z 728.597,A -85,B 0,C 180,E1 -11958.363,E2 -11958.363} C_VEL
LIN {X 0,Y 382.747,Z 737.004,A -85,B 0,C 180,E1 -11959.42,E2 -11959.42} C_VEL
LIN {X 0,Y 382.374,Z 745.398,A -85,B 0,C 180,E1 -11960.745,E2 -11960.745} C_VEL
LIN {X 0,Y 382.221,Z 752.125,A -85,B 0,C 180,E1 -11962.074,E2 -11962.074} C_VEL
LIN {X 0,Y 382.237,Z 758.383,A -85,B 0,C 180,E1 -11963.666,E2 -11963.666} C_VEL
LIN {X 0,Y 382.287,Z 763.013,A -85,B 0,C 180,E1 -11965.255,E2 -11965.255} C_VEL
LIN {X 0,Y 382.428,Z 766.224,A -85,B 0,C 180,E1 -11966.84,E2 -11966.84} C_VEL
LIN {X 0,Y 382.462,Z 767.625,A -85,B 0,C 180,E1 -11967.894,E2 -11967.894} C_VEL
LIN {X 0,Y 382.522,Z 768.481,A -85,B 0,C 180,E1 -11968.947,E2 -11968.947} C_VEL
LIN {X 0,Y 382.767,Z 768.799,A -85,B 0,C 180,E1 -11970,E2 -11970} C_VEL
LIN {X 0,Y 382.513,Z 768.528,A -85,B 0,C 180,E1 -11971.053,E2 -11971.053} C_VEL
LIN {X 0,Y 382.44,Z 767.71,A -85,B 0,C 180,E1 -11972.106,E2 -11972.106} C_VEL
LIN {X 0,Y 382.396,Z 766.386,A -85,B 0,C 180,E1 -11973.161,E2 -11973.161} C_VEL
LIN {X 0,Y 382.28,Z 763.291,A -85,B 0,C 180,E1 -11974.745,E2 -11974.745} C_VEL
LIN {X 0,Y 382.119,Z 758.872,A -85,B 0,C 180,E1 -11976.335,E2 -11976.335} C_VEL
LIN {X 0,Y 382.145,Z 752.923,A -85,B 0,C 180,E1 -11977.928,E2 -11977.928} C_VEL
LIN {X 0,Y 382.315,Z 746.646,A -85,B 0,C 180,E1 -11979.256,E2 -11979.256} C_VEL
LIN {X 0,Y 382.722,Z 738.864,A -85,B 0,C 180,E1 -11980.581,E2 -11980.581} C_VEL
LIN {X 0,Y 383.452,Z 729.154,A -85,B 0,C 180,E1 -11981.899,E2 -11981.899} C_VEL
LIN {X 0,Y 384.383,Z 717.988,A -85,B 0,C 180,E1 -11983.077,E2 -11983.077} C_VEL
LIN {X 0,Y 385.251,Z 706.699,A -85,B 0,C 180,E1 -11983.987,E2 -11983.987} C_VEL
LIN {X 0,Y 386.149,Z 694.943,A -85,B 0,C 180,E1 -11984.694,E2 -11984.694} C_VEL
LIN {X 0,Y 386.826,Z 682.8,A -85,B 0,C 180,E1 -11985.209,E2 -11985.209} C_VEL
LIN {X 0,Y 387.183,Z 664.48,A -85,B 0,C 180,E1 -11985.673,E2 -11985.673} C_VEL
LIN {X 0,Y 387.441,Z 644.681,A -85,B 0,C 180,E1 -11986.124,E2 -11986.124} C_VEL
LIN {X 0,Y 385.52,Z 615.708,A -85,B 0,C 180,E1 -11986.924,E2 -11986.924} C_VEL
LIN {X 0,Y 383.06,Z 595.279,A -85,B 0,C 180,E1 -11987.572,E2 -11987.572} C_VEL
LIN {X 0,Y 382.851,Z 593.032,A -85,B 0,C 180,E1 -11987.681,E2 -11987.681} C_VEL
LIN {X 0,Y 383.598,Z 575.003,A -85,B 0,C 180,E1 -11991.495,E2 -11991.495} C_VEL
LIN {X 0,Y 384.58,Z 558.449,A -85,B 0,C 180,E1 -11995.142,E2 -11995.142} C_VEL
LIN {X 0,Y 385.711,Z 544.69,A -85,B 0,C 180,E1 -11998.277,E2 -11998.277} C_VEL
LIN {X 0,Y 385.697,Z 541.672,A -85,B 0,C 180,E1 -11998.999,E2 -11998.999} C_VEL
LIN {X 0,Y 383.734,Z 530.942,A -85,B 0,C 180,E1 -12001.772,E2 -12001.772} C_VEL
LIN {X 0,Y 383.05,Z 527.637,A -85,B 0,C 180,E1 -12002.738,E2 -12002.738} C_VEL
LIN {X 0,Y 383.029,Z 527.586,A -85,B 0,C 180,E1 -12006.164,E2 -12006.164} C_VEL
LIN {X 0,Y 383.004,Z 527.587,A -85,B 0,C 180,E1 -12009.958,E2 -12009.958} C_VEL
LIN {X 0,Y 383,Z 527.589,A -85,B 0,C 180,E1 -12012.778,E2 -12012.778} C_VEL
LIN {X 0,Y 383.034,Z 527.583,A -85,B 0,C 180,E1 -12015.795,E2 -12015.795} C_VEL
LIN {X 0,Y 383.038,Z 527.582,A -85,B 0,C 180,E1 -12018.786,E2 -12018.786} C_VEL
LIN {X 0,Y 383.003,Z 527.586,A -85,B 0,C 180,E1 -12022.094,E2 -12022.094} C_VEL
LIN {X 0,Y 383.011,Z 527.589,A -85,B 0,C 180,E1 -12025.332,E2 -12025.332} C_VEL
LIN {X 0,Y 383.03,Z 527.581,A -85,B 0,C 180,E1 -12027.853,E2 -12027.853} C_VEL
LIN {X 0,Y 383.056,Z 527.581,A -85,B 0,C 180,E1 -12031.72,E2 -12031.72} C_VEL
LIN {X 0,Y 383.044,Z 527.587,A -85,B 0,C 180,E1 -12035.039,E2 -12035.039} C_VEL
LIN {X 0,Y 382.99,Z 527.591,A -85,B 0,C 180,E1 -12038.469,E2 -12038.469} C_VEL
LIN {X 0,Y 383.054,Z 527.579,A -85,B 0,C 180,E1 -12041.826,E2 -12041.826} C_VEL
LIN {X 0,Y 383.103,Z 527.576,A -85,B 0,C 180,E1 -12045.118,E2 -12045.118} C_VEL
LIN {X 0,Y 383.1,Z 527.578,A -85,B 0,C 180,E1 -12048.358,E2 -12048.358} C_VEL
LIN {X 0,Y 383.295,Z 527.554,A -85,B 0,C 180,E1 -12051.933,E2 -12051.933} C_VEL
LIN {X 0,Y 383.198,Z 527.566,A -85,B 0,C 180,E1 -12054.739,E2 -12054.739} C_VEL
LIN {X 0,Y 383.38,Z 527.543,A -85,B 0,C 180,E1 -12057.899,E2 -12057.899} C_VEL
LIN {X 0,Y 383.512,Z 527.527,A -85,B 0,C 180,E1 -12060,E2 -12060} C_VEL
LIN {X 0,Y 383.386,Z 527.78,A -85,B 0,C 180,E1 -12061.642,E2 -12061.642} C_VEL
LIN {X 0,Y 383.63,Z 528.782,A -85,B 0,C 180,E1 -12061.805,E2 -12061.805} C_VEL
LIN {X 0,Y 389.216,Z 542.715,A -85,B 0,C 180,E1 -12062.458,E2 -12062.458} C_VEL
LIN {X 0,Y 389.54,Z 544.786,A -85,B 0,C 180,E1 -12062.52,E2 -12062.52} C_VEL
LIN {X 0,Y 389.621,Z 565.854,A -85,B 0,C 180,E1 -12063.002,E2 -12063.002} C_VEL
LIN {X 0,Y 389.483,Z 578.131,A -85,B 0,C 180,E1 -12063.472,E2 -12063.472} C_VEL
LIN {X 0,Y 389.278,Z 590.043,A -85,B 0,C 180,E1 -12064.142,E2 -12064.142} C_VEL
LIN {X 0,Y 388.723,Z 601.237,A -85,B 0,C 180,E1 -12064.977,E2 -12064.977} C_VEL
LIN {X 0,Y 388.144,Z 611.446,A -85,B 0,C 180,E1 -12065.95,E2 -12065.95} C_VEL
LIN {X 0,Y 387.54,Z 620.6,A -85,B 0,C 180,E1 -12067.032,E2 -12067.032} C_VEL
LIN {X 0,Y 386.758,Z 629.69,A -85,B 0,C 180,E1 -12068.359,E2 -12068.359} C_VEL
LIN {X 0,Y 386.046,Z 637.307,A -85,B 0,C 180,E1 -12069.738,E2 -12069.738} C_VEL
LIN {X 0,Y 385.3,Z 644.297,A -85,B 0,C 180,E1 -12071.308,E2 -12071.308} C_VEL
LIN {X 0,Y 384.772,Z 649.088,A -85,B 0,C 180,E1 -12072.662,E2 -12072.662} C_VEL
LIN {X 0,Y 384.231,Z 653.443,A -85,B 0,C 180,E1 -12074.21,E2 -12074.21} C_VEL
LIN {X 0,Y 383.738,Z 657.025,A -85,B 0,C 180,E1 -12075.946,E2 -12075.946} C_VEL
LIN {X 0,Y 383.411,Z 659.268,A -85,B 0,C 180,E1 -12077.608,E2 -12077.608} C_VEL
LIN {X 0,Y 383.175,Z 660.45,A -85,B 0,C 180,E1 -12079.278,E2 -12079.278} C_VEL
LIN {X 0,Y 383.091,Z 660.651,A -85,B 0,C 180,E1 -12080.675,E2 -12080.675} C_VEL
LIN {X 0,Y 383.012,Z 659.635,A -85,B 0,C 180,E1 -12082.665,E2 -12082.665} C_VEL
LIN {X 0,Y 383.079,Z 658.409,A -85,B 0,C 180,E1 -12083.805,E2 -12083.805} C_VEL
LIN {X 0,Y 383.264,Z 655.607,A -85,B 0,C 180,E1 -12085.506,E2 -12085.506} C_VEL
LIN {X 0,Y 383.551,Z 651.431,A -85,B 0,C 180,E1 -12087.264,E2 -12087.264} C_VEL
LIN {X 0,Y 383.881,Z 646.065,A -85,B 0,C 180,E1 -12088.963,E2 -12088.963} C_VEL
LIN {X 0,Y 384.321,Z 639.983,A -85,B 0,C 180,E1 -12090.479,E2 -12090.479} C_VEL
LIN {X 0,Y 384.833,Z 632.503,A -85,B 0,C 180,E1 -12091.98,E2 -12091.98} C_VEL
LIN {X 0,Y 385.405,Z 623.212,A -85,B 0,C 180,E1 -12093.479,E2 -12093.479} C_VEL
LIN {X 0,Y 385.999,Z 614.764,A -85,B 0,C 180,E1 -12094.588,E2 -12094.588} C_VEL
LIN {X 0,Y 386.495,Z 604.031,A -85,B 0,C 180,E1 -12095.744,E2 -12095.744} C_VEL
LIN {X 0,Y 387.049,Z 592.29,A -85,B 0,C 180,E1 -12096.733,E2 -12096.733} C_VEL
LIN {X 0,Y 387.413,Z 581.043,A -85,B 0,C 180,E1 -12097.468,E2 -12097.468} C_VEL
LIN {X 0,Y 387.624,Z 568.205,A -85,B 0,C 180,E1 -12098.079,E2 -12098.079} C_VEL
LIN {X 0,Y 387.653,Z 554.778,A -85,B 0,C 180,E1 -12098.489,E2 -12098.489} C_VEL
LIN {X 0,Y 387.574,Z 541.893,A -85,B 0,C 180,E1 -12098.766,E2 -12098.766} C_VEL
LIN {X 0,Y 383.273,Z 528.656,A -85,B 0,C 180,E1 -12099.221,E2 -12099.221} C_VEL
LIN {X 0,Y 383.057,Z 527.689,A -85,B 0,C 180,E1 -12099.421,E2 -12099.421} C_VEL
LIN {X 0,Y 383.002,Z 527.588,A -85,B 0,C 180,E1 -12102.78,E2 -12102.78} C_VEL
LIN {X 0,Y 383.036,Z 527.583,A -85,B 0,C 180,E1 -12105.796,E2 -12105.796} C_VEL
LIN {X 0,Y 383.043,Z 527.581,A -85,B 0,C 180,E1 -12108.787,E2 -12108.787} C_VEL
LIN {X 0,Y 383.003,Z 527.586,A -85,B 0,C 180,E1 -12112.097,E2 -12112.097} C_VEL
LIN {X 0,Y 383.018,Z 527.589,A -85,B 0,C 180,E1 -12115.333,E2 -12115.333} C_VEL
LIN {X 0,Y 382.984,Z 527.59,A -85,B 0,C 180,E1 -12119.082,E2 -12119.082} C_VEL
LIN {X 0,Y 383.058,Z 527.578,A -85,B 0,C 180,E1 -12122.699,E2 -12122.699} C_VEL
LIN {X 0,Y 383.036,Z 527.582,A -85,B 0,C 180,E1 -12126.194,E2 -12126.194} C_VEL
LIN {X 0,Y 383.063,Z 527.584,A -85,B 0,C 180,E1 -12129.599,E2 -12129.599} C_VEL
LIN {X 0,Y 383.097,Z 527.574,A -85,B 0,C 180,E1 -12132.931,E2 -12132.931} C_VEL
LIN {X 0,Y 383.129,Z 527.569,A -85,B 0,C 180,E1 -12136.464,E2 -12136.464} C_VEL
LIN {X 0,Y 383.155,Z 527.566,A -85,B 0,C 180,E1 -12140.498,E2 -12140.498} C_VEL
LIN {X 0,Y 383.259,Z 527.56,A -85,B 0,C 180,E1 -12143.683,E2 -12143.683} C_VEL
LIN {X 0,Y 383.39,Z 527.542,A -85,B 0,C 180,E1 -12147.899,E2 -12147.899} C_VEL
LIN {X 0,Y 383.522,Z 527.524,A -85,B 0,C 180,E1 -12150,E2 -12150} C_VEL
LIN {X 0,Y 383.251,Z 527.555,A -85,B 0,C 180,E1 -12153.154,E2 -12153.154} C_VEL
LIN {X 0,Y 383.26,Z 527.555,A -85,B 0,C 180,E1 -12156.317,E2 -12156.317} C_VEL
LIN {X 0,Y 383.148,Z 527.57,A -85,B 0,C 180,E1 -12159.502,E2 -12159.502} C_VEL
LIN {X 0,Y 383.141,Z 527.568,A -85,B 0,C 180,E1 -12162.716,E2 -12162.716} C_VEL
LIN {X 0,Y 383.085,Z 527.581,A -85,B 0,C 180,E1 -12165.973,E2 -12165.973} C_VEL
LIN {X 0,Y 383.098,Z 527.573,A -85,B 0,C 180,E1 -12166.928,E2 -12166.928} C_VEL
LIN {X 0,Y 382.466,Z 527.658,A -85,B 0,C 180,E1 -12167.806,E2 -12167.806} C_VEL
LIN {X 0,Y 379.573,Z 528.013,A -85,B 0,C 180,E1 -12169.23,E2 -12169.23} C_VEL
LIN {X 0,Y 377.096,Z 528.323,A -85,B 0,C 180,E1 -12170.382,E2 -12170.382} C_VEL
LIN {X 0,Y 376.034,Z 528.454,A -85,B 0,C 180,E1 -12171.274,E2 -12171.274} C_VEL
LIN {X 0,Y 375.951,Z 528.466,A -85,B 0,C 180,E1 -12171.576,E2 -12171.576} C_VEL
LIN {X 0,Y 375.99,Z 528.462,A -85,B 0,C 180,E1 -12174.281,E2 -12174.281} C_VEL
LIN {X 0,Y 376.022,Z 528.455,A -85,B 0,C 180,E1 -12176.651,E2 -12176.651} C_VEL
LIN {X 0,Y 375.966,Z 528.465,A -85,B 0,C 180,E1 -12180.312,E2 -12180.312} C_VEL
LIN {X 0,Y 375.963,Z 528.468,A -85,B 0,C 180,E1 -12184.11,E2 -12184.11} C_VEL
LIN {X 0,Y 375.955,Z 528.463,A -85,B 0,C 180,E1 -12186.74,E2 -12186.74} C_VEL
LIN {X 0,Y 375.999,Z 528.463,A -85,B 0,C 180,E1 -12189.972,E2 -12189.972} C_VEL
LIN {X 0,Y 375.988,Z 528.459,A -85,B 0,C 180,E1 -12193.197,E2 -12193.197} C_VEL
LIN {X 0,Y 375.935,Z 528.466,A -85,B 0,C 180,E1 -12196.809,E2 -12196.809} C_VEL
LIN {X 0,Y 375.961,Z 528.465,A -85,B 0,C 180,E1 -12200.537,E2 -12200.537} C_VEL
LIN {X 0,Y 375.962,Z 528.463,A -85,B 0,C 180,E1 -12203.494,E2 -12203.494} C_VEL
LIN {X 0,Y 375.958,Z 528.466,A -85,B 0,C 180,E1 -12205.888,E2 -12205.888} C_VEL
LIN {X 0,Y 375.971,Z 528.462,A -85,B 0,C 180,E1 -12209.687,E2 -12209.687} C_VEL
LIN {X 0,Y 375.999,Z 528.463,A -85,B 0,C 180,E1 -12212.141,E2 -12212.141} C_VEL
LIN {X 0,Y 376.001,Z 528.461,A -85,B 0,C 180,E1 -12214.538,E2 -12214.538} C_VEL
LIN {X 0,Y 375.965,Z 528.466,A -85,B 0,C 180,E1 -12218.045,E2 -12218.045} C_VEL
LIN {X 0,Y 376.024,Z 528.454,A -85,B 0,C 180,E1 -12221.474,E2 -12221.474} C_VEL
LIN {X 0,Y 376.053,Z 528.453,A -85,B 0,C 180,E1 -12224.832,E2 -12224.832} C_VEL
LIN {X 0,Y 376.052,Z 528.455,A -85,B 0,C 180,E1 -12228.136,E2 -12228.136} C_VEL
LIN {X 0,Y 376.251,Z 528.427,A -85,B 0,C 180,E1 -12231.877,E2 -12231.877} C_VEL
LIN {X 0,Y 376.167,Z 528.441,A -85,B 0,C 180,E1 -12234.639,E2 -12234.639} C_VEL
LIN {X 0,Y 376.346,Z 528.415,A -85,B 0,C 180,E1 -12237.859,E2 -12237.859} C_VEL
LIN {X 0,Y 376.481,Z 528.399,A -85,B 0,C 180,E1 -12240,E2 -12240} C_VEL
LIN {X 0,Y 376.183,Z 528.435,A -85,B 0,C 180,E1 -12243.213,E2 -12243.213} C_VEL
LIN {X 0,Y 376.233,Z 528.434,A -85,B 0,C 180,E1 -12246.435,E2 -12246.435} C_VEL
LIN {X 0,Y 376.111,Z 528.443,A -85,B 0,C 180,E1 -12249.681,E2 -12249.681} C_VEL
LIN {X 0,Y 376.082,Z 528.447,A -85,B 0,C 180,E1 -12253.657,E2 -12253.657} C_VEL
LIN {X 0,Y 376.036,Z 528.453,A -85,B 0,C 180,E1 -12257.607,E2 -12257.607} C_VEL
LIN {X 0,Y 375.971,Z 528.466,A -85,B 0,C 180,E1 -12260.832,E2 -12260.832} C_VEL
LIN {X 0,Y 375.982,Z 528.462,A -85,B 0,C 180,E1 -12264.282,E2 -12264.282} C_VEL
LIN {X 0,Y 376.013,Z 528.462,A -85,B 0,C 180,E1 -12266.652,E2 -12266.652} C_VEL
LIN {X 0,Y 375.97,Z 528.464,A -85,B 0,C 180,E1 -12269.079,E2 -12269.079} C_VEL
LIN {X 0,Y 375.943,Z 528.471,A -85,B 0,C 180,E1 -12272.829,E2 -12272.829} C_VEL
LIN {X 0,Y 375.952,Z 528.464,A -85,B 0,C 180,E1 -12275.416,E2 -12275.416} C_VEL
LIN {X 0,Y 375.969,Z 528.463,A -85,B 0,C 180,E1 -12278.271,E2 -12278.271} C_VEL
LIN {X 0,Y 375.929,Z 528.466,A -85,B 0,C 180,E1 -12281.601,E2 -12281.601} C_VEL
LIN {X 0,Y 375.95,Z 528.466,A -85,B 0,C 180,E1 -12285.265,E2 -12285.265} C_VEL
LIN {X 0,Y 375.937,Z 528.469,A -85,B 0,C 180,E1 -12289.134,E2 -12289.134} C_VEL
LIN {X 0,Y 375.963,Z 528.462,A -85,B 0,C 180,E1 -12291.912,E2 -12291.912} C_VEL
LIN {X 0,Y 375.985,Z 528.466,A -85,B 0,C 180,E1 -12295.331,E2 -12295.331} C_VEL
LIN {X 0,Y 376.044,Z 528.713,A -85,B 0,C 180,E1 -12296.217,E2 -12296.217} C_VEL
LIN {X 0,Y 379.026,Z 543.488,A -85,B 0,C 180,E1 -12299.958,E2 -12299.958} C_VEL
LIN {X 0,Y 379.567,Z 548.783,A -85,B 0,C 180,E1 -12301.223,E2 -12301.223} C_VEL
LIN {X 0,Y 378.206,Z 564.04,A -85,B 0,C 180,E1 -12304.698,E2 -12304.698} C_VEL
LIN {X 0,Y 376.816,Z 582.462,A -85,B 0,C 180,E1 -12308.835,E2 -12308.835} C_VEL
LIN {X 0,Y 375.797,Z 601.338,A -85,B 0,C 180,E1 -12313.01,E2 -12313.01} C_VEL
LIN {X 0,Y 375.941,Z 604.19,A -85,B 0,C 180,E1 -12313.157,E2 -12313.157} C_VEL
LIN {X 0,Y 379.486,Z 647.295,A -85,B 0,C 180,E1 -12314.329,E2 -12314.329} C_VEL
LIN {X 0,Y 378.771,Z 685.109,A -85,B 0,C 180,E1 -12315.253,E2 -12315.253} C_VEL
LIN {X 0,Y 378.303,Z 697.066,A -85,B 0,C 180,E1 -12315.75,E2 -12315.75} C_VEL
LIN {X 0,Y 377.536,Z 707.968,A -85,B 0,C 180,E1 -12316.407,E2 -12316.407} C_VEL
LIN {X 0,Y 376.984,Z 717.972,A -85,B 0,C 180,E1 -12317.21,E2 -12317.21} C_VEL
LIN {X 0,Y 376.313,Z 727.122,A -85,B 0,C 180,E1 -12318.145,E2 -12318.145} C_VEL
LIN {X 0,Y 375.705,Z 735.603,A -85,B 0,C 180,E1 -12319.219,E2 -12319.219} C_VEL
LIN {X 0,Y 375.316,Z 744.082,A -85,B 0,C 180,E1 -12320.57,E2 -12320.57} C_VEL
LIN {X 0,Y 375.169,Z 750.881,A -85,B 0,C 180,E1 -12321.924,E2 -12321.924} C_VEL
LIN {X 0,Y 375.152,Z 757.19,A -85,B 0,C 180,E1 -12323.546,E2 -12323.546} C_VEL
LIN {X 0,Y 375.23,Z 761.884,A -85,B 0,C 180,E1 -12325.165,E2 -12325.165} C_VEL
LIN {X 0,Y 375.382,Z 765.131,A -85,B 0,C 180,E1 -12326.78,E2 -12326.78} C_VEL
LIN {X 0,Y 375.425,Z 766.564,A -85,B 0,C 180,E1 -12327.854,E2 -12327.854} C_VEL
LIN {X 0,Y 375.492,Z 767.432,A -85,B 0,C 180,E1 -12328.927,E2 -12328.927} C_VEL
LIN {X 0,Y 375.74,Z 767.777,A -85,B 0,C 180,E1 -12330,E2 -12330} C_VEL
LIN {X 0,Y 375.477,Z 767.517,A -85,B 0,C 180,E1 -12331.072,E2 -12331.072} C_VEL
LIN {X 0,Y 375.394,Z 766.724,A -85,B 0,C 180,E1 -12332.146,E2 -12332.146} C_VEL
LIN {X 0,Y 375.346,Z 765.42,A -85,B 0,C 180,E1 -12333.22,E2 -12333.22} C_VEL
LIN {X 0,Y 375.196,Z 762.362,A -85,B 0,C 180,E1 -12334.835,E2 -12334.835} C_VEL
LIN {X 0,Y 375.038,Z 757.965,A -85,B 0,C 180,E1 -12336.456,E2 -12336.456} C_VEL
LIN {X 0,Y 375.09,Z 752.071,A -85,B 0,C 180,E1 -12338.078,E2 -12338.078} C_VEL
LIN {X 0,Y 375.37,Z 744.425,A -85,B 0,C 180,E1 -12339.701,E2 -12339.701} C_VEL
LIN {X 0,Y 375.821,Z 736.348,A -85,B 0,C 180,E1 -12341.05,E2 -12341.05} C_VEL
LIN {X 0,Y 376.627,Z 727.418,A -85,B 0,C 180,E1 -12342.255,E2 -12342.255} C_VEL
LIN {X 0,Y 377.47,Z 717.538,A -85,B 0,C 180,E1 -12343.321,E2 -12343.321} C_VEL
LIN {X 0,Y 378.373,Z 706.566,A -85,B 0,C 180,E1 -12344.247,E2 -12344.247} C_VEL
LIN {X 0,Y 379.305,Z 695.305,A -85,B 0,C 180,E1 -12344.965,E2 -12344.965} C_VEL
LIN {X 0,Y 380.035,Z 683.338,A -85,B 0,C 180,E1 -12345.507,E2 -12345.507} C_VEL
LIN {X 0,Y 380.354,Z 670.957,A -85,B 0,C 180,E1 -12345.873,E2 -12345.873} C_VEL
LIN {X 0,Y 380.749,Z 645.136,A -85,B 0,C 180,E1 -12346.472,E2 -12346.472} C_VEL
LIN {X 0,Y 378.906,Z 616.616,A -85,B 0,C 180,E1 -12347.281,E2 -12347.281} C_VEL
LIN {X 0,Y 376.275,Z 594.722,A -85,B 0,C 180,E1 -12348.001,E2 -12348.001} C_VEL
LIN {X 0,Y 375.812,Z 591.155,A -85,B 0,C 180,E1 -12348.19,E2 -12348.19} C_VEL
LIN {X 0,Y 376.612,Z 573.998,A -85,B 0,C 180,E1 -12351.914,E2 -12351.914} C_VEL
LIN {X 0,Y 377.692,Z 557.564,A -85,B 0,C 180,E1 -12355.634,E2 -12355.634} C_VEL
LIN {X 0,Y 378.761,Z 545.148,A -85,B 0,C 180,E1 -12358.541,E2 -12358.541} C_VEL
LIN {X 0,Y 378.39,Z 540.863,A -85,B 0,C 180,E1 -12359.618,E2 -12359.618} C_VEL
LIN {X 0,Y 376.357,Z 530.334,A -85,B 0,C 180,E1 -12362.454,E2 -12362.454} C_VEL
LIN {X 0,Y 376.013,Z 528.487,A -85,B 0,C 180,E1 -12363.061,E2 -12363.061} C_VEL
LIN {X 0,Y 375.95,Z 528.469,A -85,B 0,C 180,E1 -12366.74,E2 -12366.74} C_VEL
LIN {X 0,Y 375.984,Z 528.461,A -85,B 0,C 180,E1 -12369.97,E2 -12369.97} C_VEL
LIN {X 0,Y 375.933,Z 528.468,A -85,B 0,C 180,E1 -12373.764,E2 -12373.764} C_VEL
LIN {X 0,Y 375.984,Z 528.464,A -85,B 0,C 180,E1 -12376.801,E2 -12376.801} C_VEL
LIN {X 0,Y 375.993,Z 528.46,A -85,B 0,C 180,E1 -12380.027,E2 -12380.027} C_VEL
LIN {X 0,Y 375.96,Z 528.462,A -85,B 0,C 180,E1 -12383.494,E2 -12383.494} C_VEL
LIN {X 0,Y 375.954,Z 528.466,A -85,B 0,C 180,E1 -12385.888,E2 -12385.888} C_VEL
LIN {X 0,Y 375.963,Z 528.463,A -85,B 0,C 180,E1 -12389.688,E2 -12389.688} C_VEL
LIN {X 0,Y 375.994,Z 528.461,A -85,B 0,C 180,E1 -12392.142,E2 -12392.142} C_VEL
LIN {X 0,Y 375.998,Z 528.458,A -85,B 0,C 180,E1 -12394.539,E2 -12394.539} C_VEL
LIN {X 0,Y 375.959,Z 528.465,A -85,B 0,C 180,E1 -12398.046,E2 -12398.046} C_VEL
LIN {X 0,Y 376,Z 528.459,A -85,B 0,C 180,E1 -12401.473,E2 -12401.473} C_VEL
LIN {X 0,Y 376.051,Z 528.453,A -85,B 0,C 180,E1 -12404.833,E2 -12404.833} C_VEL
LIN {X 0,Y 376.052,Z 528.455,A -85,B 0,C 180,E1 -12408.137,E2 -12408.137} C_VEL
LIN {X 0,Y 376.249,Z 528.432,A -85,B 0,C 180,E1 -12411.877,E2 -12411.877} C_VEL
LIN {X 0,Y 376.171,Z 528.441,A -85,B 0,C 180,E1 -12414.64,E2 -12414.64} C_VEL
LIN {X 0,Y 376.346,Z 528.42,A -85,B 0,C 180,E1 -12417.86,E2 -12417.86} C_VEL
LIN {X 0,Y 376.482,Z 528.403,A -85,B 0,C 180,E1 -12420,E2 -12420} C_VEL
LIN {X 0,Y 376.322,Z 528.678,A -85,B 0,C 180,E1 -12421.191,E2 -12421.191} C_VEL
LIN {X 0,Y 376.585,Z 529.802,A -85,B 0,C 180,E1 -12421.362,E2 -12421.362} C_VEL
LIN {X 0,Y 381.071,Z 540.231,A -85,B 0,C 180,E1 -12421.904,E2 -12421.904} C_VEL
LIN {X 0,Y 382.918,Z 545.161,A -85,B 0,C 180,E1 -12422.124,E2 -12422.124} C_VEL
LIN {X 0,Y 383.035,Z 568.186,A -85,B 0,C 180,E1 -12422.669,E2 -12422.669} C_VEL
LIN {X 0,Y 382.929,Z 580.257,A -85,B 0,C 180,E1 -12423.157,E2 -12423.157} C_VEL
LIN {X 0,Y 382.649,Z 592.017,A -85,B 0,C 180,E1 -12423.845,E2 -12423.845} C_VEL
LIN {X 0,Y 382.038,Z 603.526,A -85,B 0,C 180,E1 -12424.735,E2 -12424.735} C_VEL
LIN {X 0,Y 381.366,Z 614.588,A -85,B 0,C 180,E1 -12425.847,E2 -12425.847} C_VEL
LIN {X 0,Y 380.525,Z 624.874,A -85,B 0,C 180,E1 -12427.162,E2 -12427.162} C_VEL
LIN {X 0,Y 379.762,Z 633.362,A -85,B 0,C 180,E1 -12428.514,E2 -12428.514} C_VEL
LIN {X 0,Y 378.851,Z 641.578,A -85,B 0,C 180,E1 -12430.158,E2 -12430.158} C_VEL
LIN {X 0,Y 378.164,Z 648.024,A -85,B 0,C 180,E1 -12431.797,E2 -12431.797} C_VEL
LIN {X 0,Y 377.492,Z 653.103,A -85,B 0,C 180,E1 -12433.458,E2 -12433.458} C_VEL
LIN {X 0,Y 376.969,Z 656.907,A -85,B 0,C 180,E1 -12435.13,E2 -12435.13} C_VEL
LIN {X 0,Y 376.684,Z 658.81,A -85,B 0,C 180,E1 -12436.253,E2 -12436.253} C_VEL
LIN {X 0,Y 376.373,Z 660.604,A -85,B 0,C 180,E1 -12437.769,E2 -12437.769} C_VEL
LIN {X 0,Y 376.149,Z 661.658,A -85,B 0,C 180,E1 -12439.653,E2 -12439.653} C_VEL
LIN {X 0,Y 376.047,Z 661.634,A -85,B 0,C 180,E1 -12440.863,E2 -12440.863} C_VEL
LIN {X 0,Y 375.986,Z 661.175,A -85,B 0,C 180,E1 -12441.953,E2 -12441.953} C_VEL
LIN {X 0,Y 376.04,Z 659.555,A -85,B 0,C 180,E1 -12443.686,E2 -12443.686} C_VEL
LIN {X 0,Y 376.222,Z 656.766,A -85,B 0,C 180,E1 -12445.446,E2 -12445.446} C_VEL
LIN {X 0,Y 376.53,Z 652.687,A -85,B 0,C 180,E1 -12447.213,E2 -12447.213} C_VEL
LIN {X 0,Y 376.871,Z 647.167,A -85,B 0,C 180,E1 -12449.004,E2 -12449.004} C_VEL
LIN {X 0,Y 377.357,Z 640.704,A -85,B 0,C 180,E1 -12450.638,E2 -12450.638} C_VEL
LIN {X 0,Y 377.828,Z 633.97,A -85,B 0,C 180,E1 -12452.015,E2 -12452.015} C_VEL
LIN {X 0,Y 378.391,Z 625.198,A -85,B 0,C 180,E1 -12453.475,E2 -12453.475} C_VEL
LIN {X 0,Y 379.055,Z 615.694,A -85,B 0,C 180,E1 -12454.76,E2 -12454.76} C_VEL
LIN {X 0,Y 379.584,Z 605.033,A -85,B 0,C 180,E1 -12455.926,E2 -12455.926} C_VEL
LIN {X 0,Y 380.137,Z 593.287,A -85,B 0,C 180,E1 -12456.932,E2 -12456.932} C_VEL
LIN {X 0,Y 380.528,Z 581.659,A -85,B 0,C 180,E1 -12457.703,E2 -12457.703} C_VEL
LIN {X 0,Y 380.722,Z 568.956,A -85,B 0,C 180,E1 -12458.312,E2 -12458.312} C_VEL
LIN {X 0,Y 380.77,Z 556.07,A -85,B 0,C 180,E1 -12458.713,E2 -12458.713} C_VEL
LIN {X 0,Y 380.626,Z 543.058,A -85,B 0,C 180,E1 -12458.998,E2 -12458.998} C_VEL
LIN {X 0,Y 376.227,Z 529.579,A -85,B 0,C 180,E1 -12459.472,E2 -12459.472} C_VEL
LIN {X 0,Y 376.01,Z 528.571,A -85,B 0,C 180,E1 -12459.674,E2 -12459.674} C_VEL
LIN {X 0,Y 375.935,Z 528.471,A -85,B 0,C 180,E1 -12463.191,E2 -12463.191} C_VEL
LIN {X 0,Y 375.987,Z 528.46,A -85,B 0,C 180,E1 -12466.803,E2 -12466.803} C_VEL
LIN {X 0,Y 375.998,Z 528.458,A -85,B 0,C 180,E1 -12470.028,E2 -12470.028} C_VEL
LIN {X 0,Y 375.965,Z 528.468,A -85,B 0,C 180,E1 -12473.496,E2 -12473.496} C_VEL
LIN {X 0,Y 375.96,Z 528.465,A -85,B 0,C 180,E1 -12475.89,E2 -12475.89} C_VEL
LIN {X 0,Y 375.966,Z 528.466,A -85,B 0,C 180,E1 -12479.688,E2 -12479.688} C_VEL
LIN {X 0,Y 375.998,Z 528.458,A -85,B 0,C 180,E1 -12482.142,E2 -12482.142} C_VEL
LIN {X 0,Y 376.008,Z 528.456,A -85,B 0,C 180,E1 -12484.54,E2 -12484.54} C_VEL
LIN {X 0,Y 375.968,Z 528.463,A -85,B 0,C 180,E1 -12488.047,E2 -12488.047} C_VEL
LIN {X 0,Y 376.006,Z 528.462,A -85,B 0,C 180,E1 -12491.474,E2 -12491.474} C_VEL
LIN {X 0,Y 376.062,Z 528.45,A -85,B 0,C 180,E1 -12494.833,E2 -12494.833} C_VEL
LIN {X 0,Y 376.053,Z 528.452,A -85,B 0,C 180,E1 -12498.137,E2 -12498.137} C_VEL
LIN {X 0,Y 376.198,Z 528.436,A -85,B 0,C 180,E1 -12501.946,E2 -12501.946} C_VEL
LIN {X 0,Y 376.163,Z 528.437,A -85,B 0,C 180,E1 -12504.64,E2 -12504.64} C_VEL
LIN {X 0,Y 376.356,Z 528.418,A -85,B 0,C 180,E1 -12507.86,E2 -12507.86} C_VEL
LIN {X 0,Y 376.492,Z 528.4,A -85,B 0,C 180,E1 -12510,E2 -12510} C_VEL
LIN {X 0,Y 376.189,Z 528.435,A -85,B 0,C 180,E1 -12513.213,E2 -12513.213} C_VEL
LIN {X 0,Y 376.218,Z 528.431,A -85,B 0,C 180,E1 -12516.435,E2 -12516.435} C_VEL
LIN {X 0,Y 376.118,Z 528.448,A -85,B 0,C 180,E1 -12519.681,E2 -12519.681} C_VEL
LIN {X 0,Y 376.093,Z 528.45,A -85,B 0,C 180,E1 -12523.657,E2 -12523.657} C_VEL
LIN {X 0,Y 376.048,Z 528.455,A -85,B 0,C 180,E1 -12527.607,E2 -12527.607} C_VEL
LIN {X 0,Y 375.981,Z 528.46,A -85,B 0,C 180,E1 -12530.831,E2 -12530.831} C_VEL
LIN {X 0,Y 375.951,Z 528.466,A -85,B 0,C 180,E1 -12531.576,E2 -12531.576} C_VEL
LIN {X 0,Y 375.302,Z 528.553,A -85,B 0,C 180,E1 -12532.471,E2 -12532.471} C_VEL
LIN {X 0,Y 372.493,Z 528.908,A -85,B 0,C 180,E1 -12533.926,E2 -12533.926} C_VEL
LIN {X 0,Y 370.105,Z 529.203,A -85,B 0,C 180,E1 -12535.103,E2 -12535.103} C_VEL
LIN {X 0,Y 369.074,Z 529.326,A -85,B 0,C 180,E1 -12536.013,E2 -12536.013} C_VEL
LIN {X 0,Y 368.986,Z 529.334,A -85,B 0,C 180,E1 -12536.321,E2 -12536.321} C_VEL
LIN {X 0,Y 368.916,Z 529.343,A -85,B 0,C 180,E1 -12539.69,E2 -12539.69} C_VEL
LIN {X 0,Y 368.9,Z 529.342,A -85,B 0,C 180,E1 -12543.043,E2 -12543.043} C_VEL
LIN {X 0,Y 368.919,Z 529.344,A -85,B 0,C 180,E1 -12546.196,E2 -12546.196} C_VEL
LIN {X 0,Y 368.908,Z 529.341,A -85,B 0,C 180,E1 -12548.952,E2 -12548.952} C_VEL
LIN {X 0,Y 368.951,Z 529.342,A -85,B 0,C 180,E1 -12552.021,E2 -12552.021} C_VEL
LIN {X 0,Y 368.923,Z 529.339,A -85,B 0,C 180,E1 -12555.182,E2 -12555.182} C_VEL
LIN {X 0,Y 368.881,Z 529.351,A -85,B 0,C 180,E1 -12558.177,E2 -12558.177} C_VEL
LIN {X 0,Y 368.907,Z 529.341,A -85,B 0,C 180,E1 -12561.358,E2 -12561.358} C_VEL
LIN {X 0,Y 368.933,Z 529.338,A -85,B 0,C 180,E1 -12565.146,E2 -12565.146} C_VEL
LIN {X 0,Y 368.925,Z 529.339,A -85,B 0,C 180,E1 -12569.046,E2 -12569.046} C_VEL
LIN {X 0,Y 368.984,Z 529.332,A -85,B 0,C 180,E1 -12571.564,E2 -12571.564} C_VEL
LIN {X 0,Y 368.952,Z 529.335,A -85,B 0,C 180,E1 -12575.224,E2 -12575.224} C_VEL
LIN {X 0,Y 368.965,Z 529.334,A -85,B 0,C 180,E1 -12578.959,E2 -12578.959} C_VEL
LIN {X 0,Y 368.986,Z 529.337,A -85,B 0,C 180,E1 -12582.256,E2 -12582.256} C_VEL
LIN {X 0,Y 369.031,Z 529.331,A -85,B 0,C 180,E1 -12586.227,E2 -12586.227} C_VEL
LIN {X 0,Y 369.065,Z 529.325,A -85,B 0,C 180,E1 -12590.131,E2 -12590.131} C_VEL
LIN {X 0,Y 369.182,Z 529.313,A -85,B 0,C 180,E1 -12592.342,E2 -12592.342} C_VEL
LIN {X 0,Y 369.139,Z 529.318,A -85,B 0,C 180,E1 -12594.537,E2 -12594.537} C_VEL
LIN {X 0,Y 369.311,Z 529.291,A -85,B 0,C 180,E1 -12597.818,E2 -12597.818} C_VEL
LIN {X 0,Y 369.45,Z 529.275,A -85,B 0,C 180,E1 -12600,E2 -12600} C_VEL
LIN {X 0,Y 369.311,Z 529.294,A -85,B 0,C 180,E1 -12602.181,E2 -12602.181} C_VEL
LIN {X 0,Y 369.193,Z 529.312,A -85,B 0,C 180,E1 -12606.558,E2 -12606.558} C_VEL
LIN {X 0,Y 369.113,Z 529.32,A -85,B 0,C 180,E1 -12608.761,E2 -12608.761} C_VEL
LIN {X 0,Y 368.997,Z 529.331,A -85,B 0,C 180,E1 -12612.093,E2 -12612.093} C_VEL
LIN {X 0,Y 368.99,Z 529.331,A -85,B 0,C 180,E1 -12615.465,E2 -12615.465} C_VEL
LIN {X 0,Y 368.975,Z 529.336,A -85,B 0,C 180,E1 -12618.893,E2 -12618.893} C_VEL
LIN {X 0,Y 368.917,Z 529.343,A -85,B 0,C 180,E1 -12622.396,E2 -12622.396} C_VEL
LIN {X 0,Y 368.993,Z 529.331,A -85,B 0,C 180,E1 -12625.98,E2 -12625.98} C_VEL
LIN {X 0,Y 368.961,Z 529.34,A -85,B 0,C 180,E1 -12628.814,E2 -12628.814} C_VEL
LIN {X 0,Y 368.892,Z 529.344,A -85,B 0,C 180,E1 -12632.238,E2 -12632.238} C_VEL
LIN {X 0,Y 368.923,Z 529.343,A -85,B 0,C 180,E1 -12635.002,E2 -12635.002} C_VEL
LIN {X 0,Y 368.904,Z 529.346,A -85,B 0,C 180,E1 -12638.641,E2 -12638.641} C_VEL
LIN {X 0,Y 368.876,Z 529.345,A -85,B 0,C 180,E1 -12642.01,E2 -12642.01} C_VEL
LIN {X 0,Y 368.903,Z 529.345,A -85,B 0,C 180,E1 -12645.181,E2 -12645.181} C_VEL
LIN {X 0,Y 368.879,Z 529.345,A -85,B 0,C 180,E1 -12648.178,E2 -12648.178} C_VEL
LIN {X 0,Y 368.907,Z 529.343,A -85,B 0,C 180,E1 -12651.36,E2 -12651.36} C_VEL
LIN {X 0,Y 368.94,Z 529.344,A -85,B 0,C 180,E1 -12655.148,E2 -12655.148} C_VEL
LIN {X 0,Y 368.996,Z 529.515,A -85,B 0,C 180,E1 -12655.981,E2 -12655.981} C_VEL
LIN {X 0,Y 371.731,Z 543.316,A -85,B 0,C 180,E1 -12659.567,E2 -12659.567} C_VEL
LIN {X 0,Y 372.564,Z 548.862,A -85,B 0,C 180,E1 -12660.939,E2 -12660.939} C_VEL
LIN {X 0,Y 371.283,Z 562.816,A -85,B 0,C 180,E1 -12664.192,E2 -12664.192} C_VEL
LIN {X 0,Y 370.046,Z 577.949,A -85,B 0,C 180,E1 -12667.676,E2 -12667.676} C_VEL
LIN {X 0,Y 369.053,Z 594.262,A -85,B 0,C 180,E1 -12671.399,E2 -12671.399} C_VEL
LIN {X 0,Y 368.75,Z 600.392,A -85,B 0,C 180,E1 -12672.755,E2 -12672.755} C_VEL
LIN {X 0,Y 370.147,Z 617.556,A -85,B 0,C 180,E1 -12673.278,E2 -12673.278} C_VEL
LIN {X 0,Y 372.515,Z 648.156,A -85,B 0,C 180,E1 -12674.131,E2 -12674.131} C_VEL
LIN {X 0,Y 371.819,Z 684.17,A -85,B 0,C 180,E1 -12675.041,E2 -12675.041} C_VEL
LIN {X 0,Y 371.325,Z 696.049,A -85,B 0,C 180,E1 -12675.547,E2 -12675.547} C_VEL
LIN {X 0,Y 370.488,Z 707.881,A -85,B 0,C 180,E1 -12676.284,E2 -12676.284} C_VEL
LIN {X 0,Y 369.933,Z 717.636,A -85,B 0,C 180,E1 -12677.102,E2 -12677.102} C_VEL
LIN {X 0,Y 369.163,Z 727.835,A -85,B 0,C 180,E1 -12678.191,E2 -12678.191} C_VEL
LIN {X 0,Y 368.605,Z 735.956,A -85,B 0,C 180,E1 -12679.287,E2 -12679.287} C_VEL
LIN {X 0,Y 368.233,Z 744.191,A -85,B 0,C 180,E1 -12680.664,E2 -12680.664} C_VEL
LIN {X 0,Y 368.073,Z 751.875,A -85,B 0,C 180,E1 -12682.319,E2 -12682.319} C_VEL
LIN {X 0,Y 368.095,Z 757.694,A -85,B 0,C 180,E1 -12683.972,E2 -12683.972} C_VEL
LIN {X 0,Y 368.26,Z 761.974,A -85,B 0,C 180,E1 -12685.622,E2 -12685.622} C_VEL
LIN {X 0,Y 368.336,Z 764.004,A -85,B 0,C 180,E1 -12686.719,E2 -12686.719} C_VEL
LIN {X 0,Y 368.39,Z 765.479,A -85,B 0,C 180,E1 -12687.813,E2 -12687.813} C_VEL
LIN {X 0,Y 368.464,Z 766.367,A -85,B 0,C 180,E1 -12688.907,E2 -12688.907} C_VEL
LIN {X 0,Y 368.712,Z 766.749,A -85,B 0,C 180,E1 -12690,E2 -12690} C_VEL
LIN {X 0,Y 368.441,Z 766.502,A -85,B 0,C 180,E1 -12691.093,E2 -12691.093} C_VEL
LIN {X 0,Y 368.346,Z 765.741,A -85,B 0,C 180,E1 -12692.187,E2 -12692.187} C_VEL
LIN {X 0,Y 368.296,Z 764.45,A -85,B 0,C 180,E1 -12693.282,E2 -12693.282} C_VEL
LIN {X 0,Y 368.1,Z 761.43,A -85,B 0,C 180,E1 -12694.929,E2 -12694.929} C_VEL
LIN {X 0,Y 367.92,Z 756.886,A -85,B 0,C 180,E1 -12696.637,E2 -12696.637} C_VEL
LIN {X 0,Y 368.012,Z 751.216,A -85,B 0,C 180,E1 -12698.234,E2 -12698.234} C_VEL
LIN {X 0,Y 368.329,Z 743.672,A -85,B 0,C 180,E1 -12699.888,E2 -12699.888} C_VEL
LIN {X 0,Y 368.846,Z 735.707,A -85,B 0,C 180,E1 -12701.262,E2 -12701.262} C_VEL
LIN {X 0,Y 369.678,Z 726.91,A -85,B 0,C 180,E1 -12702.489,E2 -12702.489} C_VEL
LIN {X 0,Y 370.676,Z 715.799,A -85,B 0,C 180,E1 -12703.709,E2 -12703.709} C_VEL
LIN {X 0,Y 371.687,Z 704.655,A -85,B 0,C 180,E1 -12704.649,E2 -12704.649} C_VEL
LIN {X 0,Y 372.586,Z 693.366,A -85,B 0,C 180,E1 -12705.37,E2 -12705.37} C_VEL
LIN {X 0,Y 373.444,Z 680.434,A -85,B 0,C 180,E1 -12705.946,E2 -12705.946} C_VEL
LIN {X 0,Y 373.849,Z 663.286,A -85,B 0,C 180,E1 -12706.41,E2 -12706.41} C_VEL
LIN {X 0,Y 374.09,Z 645.811,A -85,B 0,C 180,E1 -12706.832,E2 -12706.832} C_VEL
LIN {X 0,Y 372.403,Z 618.109,A -85,B 0,C 180,E1 -12707.645,E2 -12707.645} C_VEL
LIN {X 0,Y 369.854,Z 596.42,A -85,B 0,C 180,E1 -12708.382,E2 -12708.382} C_VEL
LIN {X 0,Y 368.792,Z 589.596,A -85,B 0,C 180,E1 -12708.675,E2 -12708.675} C_VEL
LIN {X 0,Y 369.297,Z 579.375,A -85,B 0,C 180,E1 -12710.905,E2 -12710.905} C_VEL
LIN {X 0,Y 370.445,Z 561.694,A -85,B 0,C 180,E1 -12714.968,E2 -12714.968} C_VEL
LIN {X 0,Y 371.745,Z 546.854,A -85,B 0,C 180,E1 -12718.512,E2 -12718.512} C_VEL
LIN {X 0,Y 371.545,Z 542.861,A -85,B 0,C 180,E1 -12719.528,E2 -12719.528} C_VEL
LIN {X 0,Y 369.767,Z 533.284,A -85,B 0,C 180,E1 -12722.152,E2 -12722.152} C_VEL
LIN {X 0,Y 368.956,Z 529.372,A -85,B 0,C 180,E1 -12723.353,E2 -12723.353} C_VEL
LIN {X 0,Y 368.898,Z 529.347,A -85,B 0,C 180,E1 -12726.855,E2 -12726.855} C_VEL
LIN {X 0,Y 368.906,Z 529.343,A -85,B 0,C 180,E1 -12730.369,E2 -12730.369} C_VEL
LIN {X 0,Y 368.885,Z 529.347,A -85,B 0,C 180,E1 -12733.617,E2 -12733.617} C_VEL
LIN {X 0,Y 368.935,Z 529.344,A -85,B 0,C 180,E1 -12736.703,E2 -12736.703} C_VEL
LIN {X 0,Y 368.947,Z 529.339,A -85,B 0,C 180,E1 -12739.635,E2 -12739.635} C_VEL
LIN {X 0,Y 368.901,Z 529.344,A -85,B 0,C 180,E1 -12743.143,E2 -12743.143} C_VEL
LIN {X 0,Y 368.892,Z 529.348,A -85,B 0,C 180,E1 -12746.462,E2 -12746.462} C_VEL
LIN {X 0,Y 368.917,Z 529.34,A -85,B 0,C 180,E1 -12750.31,E2 -12750.31} C_VEL
LIN {X 0,Y 368.974,Z 529.33,A -85,B 0,C 180,E1 -12753.535,E2 -12753.535} C_VEL
LIN {X 0,Y 368.958,Z 529.336,A -85,B 0,C 180,E1 -12756.421,E2 -12756.421} C_VEL
LIN {X 0,Y 368.928,Z 529.338,A -85,B 0,C 180,E1 -12759.947,E2 -12759.947} C_VEL
LIN {X 0,Y 368.967,Z 529.338,A -85,B 0,C 180,E1 -12763.399,E2 -12763.399} C_VEL
LIN {X 0,Y 369.052,Z 529.326,A -85,B 0,C 180,E1 -12766.79,E2 -12766.79} C_VEL
LIN {X 0,Y 369.064,Z 529.327,A -85,B 0,C 180,E1 -12770.132,E2 -12770.132} C_VEL
LIN {X 0,Y 369.18,Z 529.314,A -85,B 0,C 180,E1 -12772.343,E2 -12772.343} C_VEL
LIN {X 0,Y 369.143,Z 529.316,A -85,B 0,C 180,E1 -12774.538,E2 -12774.538} C_VEL
